FUNCTION_BLOCK FB_SIS_MsgManager_6_0 IMPLEMENTS ITF_MFCS
(**************************************************************************************
 * 	Application		:	BoxControl Framework
 *	Revision		:	$Revision: 404529 $
 *	Revision date	:	$Date: 2018-04-23 08:21:38 +0200 (Mo., 23 Apr 2018) $
 *	Last changed by	:	$Author: b7bolm $
 *	URL				:	$URL: http://almscdc.swisslog.com/repo/SWPD/Development/BoxControlFramework/20_Release/trunk/01_Software/BCF/BCF/JumpStart/20_Product/10_App/11_Com/10_Lib/10_Conv/12_MFCS/11_SIS/FB_SIS_MsgManager_6_0.TcPOU $
 *
 *	Purpose			:	SIS Manager V6.0
 *
 * ------------------------------------------------------------------------------------
 *	Copyright Swisslog [IP AG], Switzerland. All rights reserved.
 * 
 * ------------------------------------------------------------------------------------
 *	
 * 	Revision History: 
 *
 * 	VERSION			DATE			INITIALS			DESCRIPTION
 *	0.1				01.01.2001		swl					Example
 *
 **************************************************************************************)
VAR_INPUT
	Config				: ST_CFG_SIS_MsgManager_6_0; // Configuration
END_VAR

VAR
	Init				: BOOL := FALSE; // Instance initialized	
	RecvTelegram		: ARRAY [1..MAX_APP_DATA_LENGTH] OF BYTE; // Last telegram read from base drive
	SendTelegram		: ARRAY [1..MAX_APP_DATA_LENGTH] OF BYTE; // Last telegram read from base drive
	fbDebugMsg			: FB_DebugMsg; // Debug Messages
	DebugMsg			: STRING(MAX_STRING_LENGTH); // String to compose the logmessage
	fbBaseDriver		: FB_SIS_BaseDriver; // Base SIS driver
	TelegramType		: STRING(3); // SIS Telegram type from the incoming message
	eMsgType			: E_ITC_MsgTypeConv;
	ReceivedLength		: UDINT; // Received length
	WritePointer		: UDINT; // Write pointer to assembly data
	
	TTA					: ST_TTA_6_0; // Struct TTA IN
	TTA_ITC				: ST_ITC_TTA; // Struct TTA IN
	TDQ					: ST_TDQ_6_0; // Struct TDQ IN
	TDQ_ITC				: ST_ITC_TDQ; // Struct TDQ IN
	SCQ					: ST_SCQ_6_0; // Struct SCQ IN
	SCQ_ITC				: ST_ITC_SCQ; // Struct SCQ IN
	GCQ					: ST_GCQ_6_0; // Struct GCQ IN
	GCQ_ITC				: ST_ITC_GCQ; // Struct ECQ IN
	ECQ					: ST_ECQ_6_0; // Struct ECQ IN
	ECQ_ITC				: ST_ITC_ECQ; // Struct ECQ IN
	FCQ					: ST_FCQ_6_0; // Struct FCQ IN
	FCQ_ITC				: ST_ITC_FCQ; // Struct FCQ IN
	SSQ					: ST_SSQ_6_0; // Struct SSQ IN
	SSQ_ITC				: ST_ITC_SSQ; // Struct SSQ IN
	GSQ					: ST_GSQ_6_0; // Struct GSQ IN
	GSQ_ITC				: ST_ITC_GSQ; // Struct GSQ IN
	ESQ					: ST_ESQ_6_0; // Struct ESQ IN
	ESQ_ITC				: ST_ITC_ESQ; // Struct ESQ IN
	FSQ					: ST_FSQ_6_0; // Struct FSQ IN
	FSQ_ITC				: ST_ITC_FSQ; // Struct FSQ IN
	TUQ					: ST_TUQ_6_0; // Struct TUQ IN
	TUQ_ITC				: ST_ITC_TUQ; // Struct TUQ IN
	SIQ					: ST_SIQ_6_0; // Struct SIQ IN
	SIQ_ITC				: ST_ITC_SIQ; // Struct SIQ IN
	MCQ					: ST_MCQ_6_0; // Struct MCQ IN
	MCQ_ITC				: ST_ITC_MCQ; // Struct MCQ IN
	DIQ					: ST_DIQ_6_0; // Struct DIQ IN
	DIQ_ITC				: ST_ITC_DIQ; // Struct DIQ IN
	SDO					: ST_SDO_6_0; // Struct SDO IN
	SDO_ITC				: ST_ITC_SDO; // Struct SDO IN
	IRQ					: ST_IRQ_6_0; // Struct IRQ IN
	IRQ_ITC				: ST_ITC_IRQ; // Struct IRQ IN
	GVQ					: ST_GVQ_6_0; // Struct GVQ IN
	GVQ_ITC				: ST_ITC_GVQ; // Struct GVQ IN
	ECR					: ST_ECR_6_0; // Struct ECR OUT
	ECR_ITC				: ST_ITC_ECR; // Struct ECR OUT
	ESR					: ST_ESR_6_0; // Struct ESR OUT
	ESR_ITC				: ST_ITC_ESR; // Struct ESR ITC
	GCR					: ST_GCR_6_0; // Struct GCR OUT
	GCR_ITC				: ST_ITC_GCR; // Struct GCR ITC
	GSR					: ST_GSR_6_0; // Struct GSR OUT
	GSR_ITC				: ST_ITC_GSR; // Struct GSR ITC
	GVR					: ST_GVR_6_0; // Struct GVR OUT
	GVR_ITC				: ST_ITC_GVR; // Struct GVR ITC
	IPR					: ST_IPR_6_0; // Struct IPR OUT
	IPR_ITC				: ST_ITC_IPR; // Struct IPR ITC
	ISR					: ST_ISR_6_0; // Struct ISR OUT
	ISR_ITC				: ST_ITC_ISR; // Struct ISR ITC
	MCR					: ST_MCR_6_0; // Struct MCR OUT
	MCR_ITC				: ST_ITC_MCR; // Struct MCR ITC
	POR					: ST_POR_6_0; // Struct POR OUT
	POR_ITC				: ST_ITC_POR; // Struct POR ITC
	SCR					: ST_SCR_6_0; // Struct SCR OUT
	SCR_ITC				: ST_ITC_SCR; // Struct SCR ITC
	SDI					: ST_SDI_6_0; // Struct SDI OUT
	SDI_ITC				: ST_ITC_SDI; // Struct SDI ITC
	SIR					: ST_SIR_6_0; // Struct SIR OUT
	SIR_ITC				: ST_ITC_SIR; // Struct SIR ITC
	SNR					: ST_SNR_6_0; // Struct SNR OUT
	SNR_ITC				: ST_ITC_SNR; // Struct SNR ITC
	SSR					: ST_SSR_6_0; // Struct SSR OUT
	SSR_ITC				: ST_ITC_SSR; // Struct SSR ITC
	TDR					: ST_TDR_6_0; // Struct TDR OUT
	TDR_ITC				: ST_ITC_TDR; // Struct TDR ITC
	TTC					: ST_TTC_6_0; // Struct TTC OUT
	TTC_ITC				: ST_ITC_TTC; // Struct TTC ITC
	TTQ					: ST_TTQ_6_0; // Struct TTQ OUT
	TTQ_ITC				: ST_ITC_TTQ; // Struct TTQ ITC
	TUR					: ST_TUR_6_0; // Struct TUR OUT
	TUR_ITC				: ST_ITC_TUR; // Struct TUR ITC
	FSR					: ST_FSR_6_0; // Struct FSR OUT
	FSR_ITC				: ST_ITC_FSR; // Struct FSR ITC
	FCR					: ST_FCR_6_0; // Struct FCR OUT
	FCR_ITC				: ST_ITC_FCR; // Struct FCR ITC
	ATR					: ST_ATR_6_0; // Struct ATR OUT
	ATR_ITC				: ST_ITC_ATR; // Struct ATR ITC
	RTR					: ST_RTR_6_0; // Struct RTR OUT
	RTR_ITC				: ST_ITC_RTR; // Struct RTR ITC
	ERR					: ST_ERR_6_0; // Struct ERR OUT
	ERR_ITC				: ST_ITC_ERR; // Struct ERR ITC
	VIQ					: ST_VIQ_6_0; // Struct VIQ OUT
	VIQ_ITC				: ST_ITC_VIQ; // Struct VIQ ITC
	VIR					: ST_VIR_6_0; // Struct VIR OUT
	VIR_ITC				: ST_ITC_VIR; // Struct VIR ITC
	RAA					: ST_RAA_6_0; // Struct RAA OUT
	RAA_ITC				: ST_ITC_RAA; // Struct RAA ITC
	RAC					: ST_RAC_6_0; // Struct RAC OUT
	RAC_ITC				: ST_ITC_RAC; // Struct RAC OUT
	RDQ					: ST_RDQ_6_0; // Struct RDQ OUT
	RDQ_ITC				: ST_ITC_RDQ; // Struct RDQ OUT
	RDR					: ST_RDR_6_0; // Struct RDR OUT
	RDR_ITC				: ST_ITC_RDR; // Struct RDR ITC
	DAQ					: ST_DAQ_6_0; // Struct DAQ IN
	DAQ_ITC				: ST_ITC_DAQ; // Struct DAQ IN
	GDQ					: ST_GDQ_6_0; // Struct GDQ IN
	GDQ_ITC				: ST_ITC_GDQ; // Struct GDQ IN
	DAR					: ST_DAR_6_0; // Struct DAR OUT
	DAR_ITC				: ST_ITC_DAR; // Struct DAR ITC
	GDR					: ST_GDR_6_0; // Struct GDR OUT
	GDR_ITC				: ST_ITC_GDR; // Struct GDR ITC
	
	
	ECR_String			: T_MaxString; // String
	ESR_String			: T_MaxString; // String
	GCR_String			: T_MaxString; // String
	GSR_String			: T_MaxString; // String
	GVR_String			: T_MaxString; // String
	IPR_String			: T_MaxString; // String
	ISR_String			: T_MaxString; // String
	MCR_String			: T_MaxString; // String
	POR_String			: T_MaxString; // String
	SCR_String			: T_MaxString; // String
	SDI_String			: T_MaxString; // String
	SIR_String			: T_MaxString; // String
	SNR_String			: T_MaxString; // String
	SSR_String			: T_MaxString; // String
	TDR_String			: T_MaxString; // String
	TTC_String			: T_MaxString; // String
	TTQ_String			: T_MaxString; // String
	TUR_String			: T_MaxString; // String
	FSR_String			: T_MaxString; // String
	FCR_String			: T_MaxString; // String
	ATR_String			: T_MaxString; // String
	RTR_String			: T_MaxString; // String
	ERR_String			: T_MaxString; // String
	VIR_String			: T_MaxString; // String
	DAR_String			: T_MaxString; // String
	GDR_String			: T_MaxString; // String
	
	// Robot telegrams
	RCQ_String			: T_MaxString; // String
	RCA_String			: T_MaxString; // String
	RCC_String			: T_MaxString; // String
	RDQ_String			: T_MaxString; // String
	RDR_String			: T_MaxString; // String
	
	Idx					: INT; // Iterator
	TempInt				: INT; // Temporary integer
	IdxOffset			: INT; // Offset telegram length
	NoError				: BOOL; // Temporary no error bit
	BufferWarningActive : BOOL; // Buffer warning level active
	BufferAlarmActive 	: BOOL; // Buffer alarm level active
END_VAR

VAR PERSISTENT
	Settings			: ST_CFG_SIS_MsgManager_6_0; // Active configuration
END_VAR

VAR CONSTANT
	MAX_APP_DATA_LENGTH	: UDINT := 30000;
END_VAR

(**************************************************************************************************************
   SIS Manager - Body never called!
***************************************************************************************************************)
;

ACTION A_PutDAQ:
(**************************************************************************************
 * 	NAME		A_PutDAQ
 * 	FUNCTION	Process DAQ
 **************************************************************************************)

// Clear data structure 
MEMSET(destAddr := ADR(DAQ), fillByte := 0, n := SIZEOF(DAQ));
				
// Copy the TDQ data fields to the DAQ data structure 
IdxOffset := SIS_6_0.APP_DATA_OFFSET+1;
// Copy
MEMCPY(destAddr := ADR(DAQ.Position), srcAddr := ADR(RecvTelegram[IdxOffset]), n := INT_TO_UDINT(SIS_6_0.POSITION_STRINGLENGTH));
// Adjust index
IdxOffset := IdxOffset + SIS_6_0.POSITION_STRINGLENGTH;
// Copy
MEMCPY(destAddr := ADR(DAQ.NumberOfSets), srcAddr := ADR(RecvTelegram[IdxOffset]), n := INT_TO_UDINT(SIS_6_0.DATA_ACQUISITION_NUMBEROFSETS));
// Adjust index
IdxOffset := IdxOffset + SIS_6_0.DATA_ACQUISITION_NUMBEROFSETS;
// Copy
MEMCPY(destAddr := ADR(DAQ.Code), srcAddr := ADR(RecvTelegram[IdxOffset]), n := INT_TO_UDINT(SIS_6_0.DATA_ACQUISITION_CODE));
// Adjust index
IdxOffset := IdxOffset + SIS_6_0.DATA_ACQUISITION_CODE;

FOR Idx := 1 TO STRING_TO_INT(DAQ.NumberOfSets) DO
	
	MEMCPY(destAddr := ADR(DAQ.Variable[Idx]), srcAddr := ADR(RecvTelegram[IdxOffset]), n := INT_TO_UDINT(SIS_6_0.DATA_ACQUISITION_VARIABLENAME));
 
	IdxOffset := IdxOffset + SIS_6_0.DATA_ACQUISITION_VARIABLENAME;
	// Copy
	MEMCPY(destAddr := ADR(DAQ.MaxReportTime[Idx]), srcAddr := ADR(RecvTelegram[IdxOffset]), n := INT_TO_UDINT(SIS_6_0.DATA_ACQUISITION_MAXREPORTTIME));
   // Adjust index
	IdxOffset := IdxOffset + SIS_6_0.DATA_ACQUISITION_MAXREPORTTIME;
	// Copy
	MEMCPY(destAddr := ADR(DAQ.SampleTime[Idx]), srcAddr := ADR(RecvTelegram[IdxOffset]), n := INT_TO_UDINT(SIS_6_0.DATA_ACQUISITION_SAMPLETIME));
	 // Adjust index
	IdxOffset := IdxOffset + SIS_6_0.DATA_ACQUISITION_SAMPLETIME;
	// Copy
	MEMCPY(destAddr := ADR(DAQ.Threshold[Idx]), srcAddr := ADR(RecvTelegram[IdxOffset]), n := INT_TO_UDINT(SIS_6_0.DATA_ACQUISITION_THRESHOLD));
	 // Adjust index
	IdxOffset := IdxOffset + SIS_6_0.DATA_ACQUISITION_THRESHOLD;
	// Copy
	MEMCPY(destAddr := ADR(DAQ.Option[Idx]), srcAddr := ADR(RecvTelegram[IdxOffset]), n := INT_TO_UDINT(SIS_6_0.DATA_ACQUISITION_BIT));
	 // Adjust index
	IdxOffset := IdxOffset + SIS_6_0.DATA_ACQUISITION_BIT;
	// Copy
	MEMCPY(destAddr := ADR(DAQ.Enable[Idx]), srcAddr := ADR(RecvTelegram[IdxOffset]), n := INT_TO_UDINT(SIS_6_0.DATA_ACQUISITION_BIT));
	
	IdxOffset := IdxOffset + SIS_6_0.DATA_ACQUISITION_BIT;
	
END_FOR



// Map to ITC
DAQ_ITC.Position :=  DAQ.Position;
DAQ_ITC.Code := STRING_TO_INT(DAQ.Code);
DAQ_ITC.NumberOfSets := STRING_TO_INT(DAQ.NumberOfSets);

FOR Idx := 1 TO STRING_TO_INT(DAQ.NumberOfSets) DO

	DAQ_ITC.Set[Idx].mVariableName := DAQ.Variable[Idx];
	DAQ_ITC.Set[Idx].MaxReportTime := F_MaxReportTime_TO_Time(sTimeIn:= DAQ.MaxReportTime[Idx]);
	DAQ_ITC.Set[Idx].SampleTime := F_SampleTime_TO_TIME(SampleTimeString:=DAQ.SampleTime[Idx]);
	DAQ_ITC.Set[Idx].Threshold := STRING_TO_INT(DAQ.Threshold[Idx]);
	DAQ_ITC.Set[Idx].Option := INT_TO_BOOL(STRING_TO_INT(DAQ.Option[Idx]));
	DAQ_ITC.Set[Idx].Enable :=  INT_TO_BOOL(STRING_TO_INT(DAQ.Enable[Idx]));
END_FOR

// Forward to mirror channel
M_MirrorData(Data := ADR(RecvTelegram), DataLen := ReceivedLength);

// Forward message to ITC
NoError := fbITC_Manager.M_AddData(
			meChannelSrc := Settings.MFCS_Channel,
			mMsgType	 := E_ITC_MsgTypeConv.DATA_ACQUISITION_REQUEST,
			mpData		 := ADR(DAQ_ITC),
			mLen		 := SIZEOF(DAQ_ITC));

// If forwarding was successful
IF NoError THEN
	// Message processed
	fbBaseDriver.M_ProcessedMsg();
ELSE	
	DebugMsg := 'DAQ - Could not be forwarded to ITC';
	fbDebugMsg.M_SendErrorMsg(DebugMsg);		
END_IF
END_ACTION

ACTION A_PutDIQ:
(**************************************************************************************
 * 	NAME		A_PutDIQ
 * 	FUNCTION	Process DIQ
 **************************************************************************************)
 
// Clear structure
MEMSET(destAddr := ADR(DIQ), fillByte := 0, n := SIZEOF(DIQ));

// Forward to mirror channel
M_MirrorData(Data := ADR(RecvTelegram), DataLen := ReceivedLength);

// Forward message to ITC
NoError := fbITC_Manager.M_AddData(
			meChannelSrc := Settings.MFCS_Channel,
			mMsgType	 := E_ITC_MsgTypeConv.DIGITAL_INPUT_REQUEST,
			mpData		 := 0,
			mLen		 := 0);

// If forwarding was successful
IF NoError THEN
	// Message processed
	fbBaseDriver.M_ProcessedMsg();
	
ELSE	
	DebugMsg := 'DIQ - Could not be forwarded to ITC';
	fbDebugMsg.M_SendErrorMsg(DebugMsg);	
END_IF
END_ACTION

ACTION A_PutECQ:
(**************************************************************************************
 * 	NAME		A_PutECQ
 * 	FUNCTION	Process ECQ
 **************************************************************************************)
 
// Clear data structure 
MEMSET(destAddr := ADR(ECQ), fillByte := 0, n := SIZEOF(ECQ));

// Copy the ECQ data fields to the ECQ data structure 
IdxOffset := SIS_6_0.APP_DATA_OFFSET + 1;

// Copy
MEMCPY(destAddr := ADR(ECQ.Position), srcAddr := ADR(RecvTelegram[IdxOffset]), n := INT_TO_UDINT(SIS_6_0.POSITION_STRINGLENGTH));
// Adjust index
IdxOffset := IdxOffset + SIS_6_0.POSITION_STRINGLENGTH;
// Copy
MEMCPY(destAddr := ADR(ECQ.Code), srcAddr := ADR(RecvTelegram[IdxOffset]), n := INT_TO_UDINT(SIS_6_0.CONTROLCODE_STRINGLENGTH));
// Adjust index
IdxOffset := IdxOffset + SIS_6_0.CONTROLCODE_STRINGLENGTH;
// Copy
MEMCPY(destAddr := ADR(ECQ.Variable), srcAddr := ADR(RecvTelegram[IdxOffset]), n := INT_TO_UDINT(SIS_6_0.CONTROLVARIABLE_STRINGLENGTH));


// Map to ITC
ECQ_ITC.Position := ECQ.Position;
ECQ_ITC.Code := STRING_TO_INT(ECQ.Code);
ECQ_ITC.Variable := STRING_TO_INT(ECQ.Variable);

// Forward to mirror channel
M_MirrorData(Data := ADR(RecvTelegram), DataLen := ReceivedLength);

// Forward message to ITC
NoError := fbITC_Manager.M_AddData(
			meChannelSrc := Settings.MFCS_Channel,
			mMsgType	 := E_ITC_MsgTypeCOnv.ELEMENT_CONTROL_REQUEST,
			mpData		 := ADR(ECQ_ITC),
			mLen		 := SIZEOF(ECQ_ITC));

	
// If forwarding was successful
IF NoError THEN
	// Message processed
	fbBaseDriver.M_ProcessedMsg();
ELSE	
	DebugMsg := 'ECQ - Could not be forwarded to ITC';
	fbDebugMsg.M_SendErrorMsg(DebugMsg);	
END_IF
END_ACTION

ACTION A_PutESQ:
(**************************************************************************************
 * 	NAME		A_PutESQ
 * 	FUNCTION	Process ESQ
 **************************************************************************************)

// Clear data structure 
MEMSET(destAddr := ADR(ESQ), fillByte := 0, n := SIZEOF(ESQ));

// Copy the ESQ data fields to the ESQ data structure 
IdxOffset := SIS_6_0.APP_DATA_OFFSET + 1;

MEMCPY(destAddr := ADR(ESQ.Position), srcAddr := ADR(RecvTelegram[IdxOffset]), n := 12);

// Map to ITC
ESQ_ITC.Position := ESQ.Position;

// Forward to mirror channel
M_MirrorData(Data := ADR(RecvTelegram), DataLen := ReceivedLength);

// Forward message to ITC
NoError := fbITC_Manager.M_AddData(
			meChannelSrc := Settings.MFCS_Channel,
			mMsgType	 := E_ITC_MsgTypeCOnv.ELEMENT_STATUS_REQUEST,
			mpData		 := ADR(ESQ_ITC),
			mLen		 := SIZEOF(ESQ_ITC));

// If forwarding was successful
IF NoError THEN
	// Message processed
	fbBaseDriver.M_ProcessedMsg();
	
ELSE	
	DebugMsg := 'ESQ - Could not be forwarded to ITC';
	fbDebugMsg.M_SendErrorMsg(DebugMsg);
END_IF
END_ACTION

ACTION A_PutFCQ:
(**************************************************************************************
 * 	NAME		A_PutFCQ
 * 	FUNCTION	Process FCQ
 **************************************************************************************)
 
// Clear data structure 
MEMSET(destAddr := ADR(FCQ), fillByte := 0, n := SIZEOF(FCQ));

// Copy the FCQ data fields to the FCQ data structure 
IdxOffset := SIS_6_0.APP_DATA_OFFSET + 1;

// Copy
MEMCPY(destAddr := ADR(FCQ.Position), srcAddr := ADR(RecvTelegram[IdxOffset]), n := INT_TO_UDINT(SIS_6_0.POSITION_STRINGLENGTH));
// Adjust index
IdxOffset := IdxOffset + SIS_6_0.POSITION_STRINGLENGTH;
// Copy
MEMCPY(destAddr := ADR(FCQ.Code), srcAddr := ADR(RecvTelegram[IdxOffset]), n := INT_TO_UDINT(SIS_6_0.CONTROLCODE_STRINGLENGTH));
// Adjust index
IdxOffset := IdxOffset + SIS_6_0.CONTROLCODE_STRINGLENGTH;
// Copy
MEMCPY(destAddr := ADR(FCQ.Variable), srcAddr := ADR(RecvTelegram[IdxOffset]), n := INT_TO_UDINT(SIS_6_0.CONTROLVARIABLE_STRINGLENGTH));

// Map to ITC
FCQ_ITC.Position := FCQ.Position; 
FCQ_ITC.Code := STRING_TO_INT(FCQ.Code);
FCQ_ITC.Variable := STRING_TO_DINT(FCQ.Variable);

// Forward to mirror channel
M_MirrorData(Data := ADR(RecvTelegram), DataLen := ReceivedLength);

// Forward message to ITC
NoError := fbITC_Manager.M_AddData(
			meChannelSrc := Settings.MFCS_Channel,
			mMsgType	 := E_ITC_MsgTypeCOnv.FUNCTION_CONTROL_REQUEST,
			mpData		 := ADR(FCQ_ITC),
			mLen		 := SIZEOF(FCQ_ITC));
	
// If forwarding was successful
IF NoError THEN
	// Message processed
	fbBaseDriver.M_ProcessedMsg();
	
ELSE	
	DebugMsg := 'FCQ - Could not be forwarded to ITC';
	fbDebugMsg.M_SendErrorMsg(DebugMsg);
END_IF
END_ACTION

ACTION A_PutFSQ:
(**************************************************************************************
 * 	NAME		A_PutFSQ
 * 	FUNCTION	Process FSQ
 **************************************************************************************)

// Clear data structure 
MEMSET(destAddr := ADR(FSQ), fillByte := 0, n := SIZEOF(FSQ));

// Copy the FSQ data fields to the FSQ data structure 
IdxOffset := SIS_6_0.APP_DATA_OFFSET + 1;
// Copy
MEMCPY(destAddr := ADR(FSQ.Position), srcAddr := ADR(RecvTelegram[IdxOffset]), n := INT_TO_UDINT(SIS_6_0.POSITION_STRINGLENGTH));

// Map to ITC
FSQ_ITC.Position := FSQ.Position; 

// Forward to mirror channel
M_MirrorData(Data := ADR(RecvTelegram), DataLen := ReceivedLength);

// Forward message to ITC
NoError := fbITC_Manager.M_AddData(
			meChannelSrc := Settings.MFCS_Channel,
			mMsgType	 := E_ITC_MsgTypeCOnv.FUNCTION_STATUS_REQUEST,
			mpData		 := ADR(FSQ_ITC),
			mLen		 := SIZEOF(FSQ_ITC));

// If forwarding was successful
IF NoError THEN
	// Message processed
	fbBaseDriver.M_ProcessedMsg();
	
ELSE	
	DebugMsg := 'FSQ - Could not be forwarded to ITC';
	fbDebugMsg.M_SendErrorMsg(DebugMsg);	
END_IF
END_ACTION

ACTION A_PutGCQ:
(**************************************************************************************
 * 	NAME		A_PutGCQ
 * 	FUNCTION	Process GCQ
 **************************************************************************************)
 
// Clear data structure 
MEMSET(destAddr := ADR(GCQ), fillByte := 0, n := SIZEOF(GCQ));

// Copy the GCQ data fields to the GCQ data structure 
IdxOffset := SIS_6_0.APP_DATA_OFFSET + 1;
// Copy
MEMCPY(destAddr := ADR(GCQ.GroupName), srcAddr := ADR(RecvTelegram[IdxOffset]), n := INT_TO_UDINT(SIS_6_0.POSITION_STRINGLENGTH));
// Adjust index
IdxOffset := IdxOffset + SIS_6_0.POSITION_STRINGLENGTH;
// Copy
MEMCPY(destAddr := ADR(GCQ.Code), srcAddr := ADR(RecvTelegram[IdxOffset]), n := INT_TO_UDINT(SIS_6_0.CONTROLCODE_STRINGLENGTH));
// Adjust index
IdxOffset := IdxOffset + SIS_6_0.CONTROLCODE_STRINGLENGTH;
// Copy
MEMCPY(destAddr := ADR(GCQ.Variable), srcAddr := ADR(RecvTelegram[IdxOffset]), n := INT_TO_UDINT(SIS_6_0.CONTROLVARIABLE_STRINGLENGTH));

// Map to ITC
GCQ_ITC.Position := GCQ.GroupName;
GCQ_ITC.Code := STRING_TO_INT(GCQ.Code);
GCQ_ITC.Variable := STRING_TO_DINT(GCQ.Variable);

// Forward to mirror channel
M_MirrorData(Data := ADR(RecvTelegram), DataLen := ReceivedLength);

// Forward message to ITC
NoError := fbITC_Manager.M_AddData(
			meChannelSrc := Settings.MFCS_Channel,
			mMsgType	 := E_ITC_MsgTypeConv.GROUP_CONTROL_REQUEST,
			mpData		 := ADR(GCQ_ITC),
			mLen		 := SIZEOF(GCQ_ITC));

// If forwarding was successful
IF NoError THEN
	// Message processed
	fbBaseDriver.M_ProcessedMsg();
	
ELSE	
	DebugMsg := 'GCQ - Could not be forwarded to ITC';
	fbDebugMsg.M_SendErrorMsg(DebugMsg);	
END_IF
END_ACTION

ACTION A_PutGDQ:
(**************************************************************************************
 * 	NAME		A_PutGDQ
 * 	FUNCTION	Process GDQ
 **************************************************************************************)

// Clear data structure 
MEMSET(destAddr := ADR(GDQ), fillByte := 0, n := SIZEOF(GDQ));

// Copy the GDQ data fields to the GDQ data structure 
IdxOffset := SIS_6_0.APP_DATA_OFFSET+1;
// Copy
MEMCPY(destAddr := ADR(GDQ.Position), srcAddr := ADR(RecvTelegram[IdxOffset]), n := INT_TO_UDINT(SIS_6_0.POSITION_STRINGLENGTH));
// Adjust index
IdxOffset := IdxOffset + SIS_6_0.POSITION_STRINGLENGTH;
// Copy
MEMCPY(destAddr := ADR(GDQ.Variable), srcAddr := ADR(RecvTelegram[IdxOffset]), n := INT_TO_UDINT(SIS_6_0.DATA_ACQUISITION_VARIABLENAME));
// Adjust index
IdxOffset := IdxOffset + SIS_6_0.DATA_ACQUISITION_VARIABLENAME;

// Map to ITC
GDQ_ITC.Position :=  GDQ.Position;
GDQ_ITC.Variable :=  GDQ.Variable;

// Forward to mirror channel
M_MirrorData(Data := ADR(RecvTelegram), DataLen := ReceivedLength);

// Forward message to ITC
NoError := fbITC_Manager.M_AddData(
			meChannelSrc := Settings.MFCS_Channel,
			mMsgType	 := E_ITC_MsgTypeConv.GATHERED_DATA_REQUEST,
			mpData		 := ADR(GDQ_ITC),
			mLen		 := SIZEOF(GDQ_ITC));

// If forwarding was successful
IF NoError THEN
	// Message processed
	fbBaseDriver.M_ProcessedMsg();
	
ELSE	
	DebugMsg := 'GDQ - Could not be forwarded to ITC';
	fbDebugMsg.M_SendErrorMsg(DebugMsg);	
END_IF
END_ACTION

ACTION A_PutGSQ:
(**************************************************************************************
 * 	NAME		A_PutGSQ
 * 	FUNCTION	Process GSQ
 **************************************************************************************)

// Clear data structure 
MEMSET(destAddr := ADR(GSQ), fillByte := 0, n := SIZEOF(GSQ));

// Copy the GSQ data fields to the GSQ data structure 
IdxOffset := SIS_6_0.APP_DATA_OFFSET + 1;

MEMCPY(destAddr := ADR(GSQ.GroupName), srcAddr := ADR(RecvTelegram[IdxOffset]), n := INT_TO_UDINT(SIS_6_0.POSITION_STRINGLENGTH));

// Map to ITC
GSQ_ITC.Position := GSQ.GroupName;

// Forward to mirror channel
M_MirrorData(Data := ADR(RecvTelegram), DataLen := ReceivedLength);

// Forward message to ITC
NoError := fbITC_Manager.M_AddData(
			meChannelSrc := Settings.MFCS_Channel,
			mMsgType	 := E_ITC_MsgTypeConv.GROUP_STATUS_REQUEST,
			mpData		 := ADR(GSQ_ITC),
			mLen		 := SIZEOF(GSQ_ITC));

// If forwarding was successful
IF NoError THEN
	// Message processed
	fbBaseDriver.M_ProcessedMsg();
	
ELSE	
	DebugMsg := 'GSQ - Could not be forwarded to ITC';
	fbDebugMsg.M_SendErrorMsg(DebugMsg);	
END_IF
END_ACTION

ACTION A_PutGVQ:
(**************************************************************************************
 * 	NAME		A_PutGVQ
 * 	FUNCTION	Process GVQ
 **************************************************************************************)

// Clear data structure 
MEMSET(destAddr := ADR(GVQ), fillByte := 0, n := SIZEOF(GVQ));

// Copy the GVQ data fields to the GVQ data structure 
IdxOffset := SIS_6_0.APP_DATA_OFFSET + 1;
// Copy
MEMCPY(destAddr := ADR(GVQ.Code), srcAddr := ADR(RecvTelegram[IdxOffset]), n := INT_TO_UDINT(SIS_6_0.GVQ_CODE_STRINGLENGTH));
// Adjust index
IdxOffset := IdxOffset + SIS_6_0.GVQ_CODE_STRINGLENGTH;
// Copy
MEMCPY(destAddr := ADR(GVQ.Number), srcAddr := ADR(RecvTelegram[IdxOffset]), n := INT_TO_UDINT(SIS_6_0.GVQ_NUMBER_STRINGLENGTH));
// Adjust index
IdxOffset := IdxOffset + SIS_6_0.GVQ_NUMBER_STRINGLENGTH;
// Copy
MEMCPY(destAddr := ADR(GVQ.Quantity), srcAddr := ADR(RecvTelegram[IdxOffset]), n := INT_TO_UDINT(SIS_6_0.GVQ_QUANTITY_STRINGLENGTH));
// Adjust index
IdxOffset := IdxOffset + SIS_6_0.GVQ_QUANTITY_STRINGLENGTH;
// Copy
MEMCPY(destAddr := ADR(GVQ.Variable[0]), srcAddr := ADR(RecvTelegram[IdxOffset]), n := INT_TO_UDINT(SIS_6_0.GVQ_VARIABLE_STRINGLENGTH));
// Adjust index
IdxOffset := IdxOffset + SIS_6_0.GVQ_VARIABLE_STRINGLENGTH;
// Copy
MEMCPY(destAddr := ADR(GVQ.Variable[1]), srcAddr := ADR(RecvTelegram[IdxOffset]), n := INT_TO_UDINT(SIS_6_0.GVQ_VARIABLE_STRINGLENGTH));
// Adjust index
IdxOffset := IdxOffset + SIS_6_0.GVQ_VARIABLE_STRINGLENGTH;
// Copy
MEMCPY(destAddr := ADR(GVQ.Variable[2]), srcAddr := ADR(RecvTelegram[IdxOffset]), n := INT_TO_UDINT(SIS_6_0.GVQ_VARIABLE_STRINGLENGTH));
// Adjust index
IdxOffset := IdxOffset + SIS_6_0.GVQ_VARIABLE_STRINGLENGTH;
// Copy
MEMCPY(destAddr := ADR(GVQ.Variable[3]), srcAddr := ADR(RecvTelegram[IdxOffset]), n := INT_TO_UDINT(SIS_6_0.GVQ_VARIABLE_STRINGLENGTH));
// Adjust index
IdxOffset := IdxOffset + SIS_6_0.GVQ_VARIABLE_STRINGLENGTH;
// Copy
MEMCPY(destAddr := ADR(GVQ.Variable[4]), srcAddr := ADR(RecvTelegram[IdxOffset]), n := INT_TO_UDINT(SIS_6_0.GVQ_VARIABLE_STRINGLENGTH));
// Adjust index
IdxOffset := IdxOffset + SIS_6_0.GVQ_VARIABLE_STRINGLENGTH;
// Copy
MEMCPY(destAddr := ADR(GVQ.Variable[5]), srcAddr := ADR(RecvTelegram[IdxOffset]), n := INT_TO_UDINT(SIS_6_0.GVQ_VARIABLE_STRINGLENGTH));
// Adjust index
IdxOffset := IdxOffset + SIS_6_0.GVQ_VARIABLE_STRINGLENGTH;
// Copy
MEMCPY(destAddr := ADR(GVQ.Variable[6]), srcAddr := ADR(RecvTelegram[IdxOffset]), n := INT_TO_UDINT(SIS_6_0.GVQ_VARIABLE_STRINGLENGTH));
// Adjust index
IdxOffset := IdxOffset + SIS_6_0.GVQ_VARIABLE_STRINGLENGTH;
// Copy
MEMCPY(destAddr := ADR(GVQ.Variable[7]), srcAddr := ADR(RecvTelegram[IdxOffset]), n := INT_TO_UDINT(SIS_6_0.GVQ_VARIABLE_STRINGLENGTH));
// Adjust index
IdxOffset := IdxOffset + SIS_6_0.GVQ_VARIABLE_STRINGLENGTH;
// Copy
MEMCPY(destAddr := ADR(GVQ.Variable[8]), srcAddr := ADR(RecvTelegram[IdxOffset]), n := INT_TO_UDINT(SIS_6_0.GVQ_VARIABLE_STRINGLENGTH));
// Adjust index
IdxOffset := IdxOffset + SIS_6_0.GVQ_VARIABLE_STRINGLENGTH;
// Copy
MEMCPY(destAddr := ADR(GVQ.Variable[9]), srcAddr := ADR(RecvTelegram[IdxOffset]), n := INT_TO_UDINT(SIS_6_0.GVQ_VARIABLE_STRINGLENGTH));

// Map to ITC
GVQ_ITC.Code := STRING_TO_INT(GVQ.Code);
GVQ_ITC.Number := STRING_TO_INT(GVQ.Number);
GVQ_ITC.Quantity := STRING_TO_INT(GVQ.Quantity);
GVQ_ITC.Variable[0] := STRING_TO_DINT(GVQ.Variable[0]);
GVQ_ITC.Variable[1] := STRING_TO_DINT(GVQ.Variable[1]);
GVQ_ITC.Variable[2] := STRING_TO_DINT(GVQ.Variable[2]);
GVQ_ITC.Variable[3] := STRING_TO_DINT(GVQ.Variable[3]);
GVQ_ITC.Variable[4] := STRING_TO_DINT(GVQ.Variable[4]);
GVQ_ITC.Variable[5] := STRING_TO_DINT(GVQ.Variable[5]);
GVQ_ITC.Variable[6] := STRING_TO_DINT(GVQ.Variable[6]);
GVQ_ITC.Variable[7] := STRING_TO_DINT(GVQ.Variable[7]);
GVQ_ITC.Variable[8] := STRING_TO_DINT(GVQ.Variable[8]);
GVQ_ITC.Variable[9] := STRING_TO_DINT(GVQ.Variable[9]);

// Forward to mirror channel
M_MirrorData(Data := ADR(RecvTelegram), DataLen := ReceivedLength);

// Forward message to ITC
NoError := fbITC_Manager.M_AddData(
			meChannelSrc := Settings.MFCS_Channel,
			mMsgType	 := E_ITC_MsgTypeConv.GLOBAL_VARIABLE_REQUEST,
			mpData		 := ADR(GVQ_ITC),
			mLen	 := SIZEOF(GVQ_ITC));
	
// If forwarding was successful
IF NoError THEN
	// Message processed
	fbBaseDriver.M_ProcessedMsg();
	
ELSE	
	DebugMsg := 'GVQ - Could not be forwarded to ITC';
	fbDebugMsg.M_SendErrorMsg(DebugMsg);	
END_IF
END_ACTION

ACTION A_PutIRQ:
(**************************************************************************************
 * 	NAME		A_PutIRQ
 * 	FUNCTION	Process IRQ
 **************************************************************************************)
 
// Clear data structure 
MEMSET(destAddr := ADR(IRQ), fillByte := 0, n := SIZEOF(IRQ));

// Copy the IRQ data fields to the IRQ data structure 
IdxOffset := SIS_6_0.APP_DATA_OFFSET + 1;
// Copy
MEMCPY(destAddr := ADR(IRQ.SignalType), srcAddr := ADR(RecvTelegram[IdxOffset]), n := INT_TO_UDINT(SIS_6_0.IRQ_SIGNALTYPE_STRINGLENGTH));
// Adjust index
IdxOffset := IdxOffset + SIS_6_0.IRQ_SIGNALTYPE_STRINGLENGTH;
// Copy
MEMCPY(destAddr := ADR(IRQ.StartSignalNumber), srcAddr := ADR(RecvTelegram[IdxOffset]), n := INT_TO_UDINT(SIS_6_0.IRQ_START_SIGNAL_NUMBER_STRINGLENGTH));
// Adjust index
IdxOffset := IdxOffset + SIS_6_0.IRQ_START_SIGNAL_NUMBER_STRINGLENGTH;
// Copy
MEMCPY(destAddr := ADR(IRQ.DataLength), srcAddr := ADR(RecvTelegram[IdxOffset]), n := INT_TO_UDINT(SIS_6_0.IRQ_DATALENGTH_STRINGLENGTH));

// Map to ITC
IRQ_ITC.DataLength := STRING_TO_INT(IRQ.DataLength);
IRQ_ITC.SignalType := STRING_TO_INT(IRQ.SignalType);
IRQ_ITC.StartSignalNumber := STRING_TO_INT(IRQ.StartSignalNumber);

// Forward to mirror channel
M_MirrorData(Data := ADR(RecvTelegram), DataLen := ReceivedLength);

// Forward message to ITC
NoError := fbITC_Manager.M_AddData(
			meChannelSrc := Settings.MFCS_Channel,
			mMsgType	 := E_ITC_MsgTypeConv.I_O_STATUS_REQUEST,
			mpData		 := ADR(IRQ_ITC),
			mLen		 := SIZEOF(IRQ_ITC));


// If forwarding was successful
IF NoError THEN
	// Message processed
	fbBaseDriver.M_ProcessedMsg();
	
ELSE	
	DebugMsg := 'IRQ - Could not be forwarded to ITC';
	fbDebugMsg.M_SendErrorMsg(DebugMsg);	
END_IF
END_ACTION

ACTION A_PutMCQ:
(**************************************************************************************
 * 	NAME		A_PutMCQ
 * 	FUNCTION	Process MCQ
 **************************************************************************************)
 
// Clear data structure 
MEMSET(destAddr := ADR(MCQ), fillByte := 0, n := SIZEOF(MCQ));

// Copy the MCQ data fields to the MCQ data structure 
IdxOffset := SIS_6_0.APP_DATA_OFFSET + 1;
// Copy
MEMCPY(destAddr := ADR(MCQ.Position), srcAddr := ADR(RecvTelegram[IdxOffset]), n := INT_TO_UDINT(SIS_6_0.POSITION_STRINGLENGTH));
// Adjust index
IdxOffset := IdxOffset + SIS_6_0.POSITION_STRINGLENGTH;
// Copy
MEMCPY(destAddr := ADR(MCQ.Code), srcAddr := ADR(RecvTelegram[IdxOffset]), n := INT_TO_UDINT(SIS_6_0.MCQ_CODE_STRINGLENGTH));
// Adjust index
IdxOffset := IdxOffset + SIS_6_0.MCQ_CODE_STRINGLENGTH;
// Copy
MEMCPY(destAddr := ADR(MCQ.Speed), srcAddr := ADR(RecvTelegram[IdxOffset]), n := INT_TO_UDINT(SIS_6_0.MCQ_SPEED_STRINGLENGTH));
// Adjust index
IdxOffset := IdxOffset + SIS_6_0.MCQ_SPEED_STRINGLENGTH;
// Copy
MEMCPY(destAddr := ADR(MCQ.Axis1Fwd), srcAddr := ADR(RecvTelegram[IdxOffset]), n := INT_TO_UDINT(SIS_6_0.MCQ_AXIS_STRINGLENGTH));
// Adjust index
IdxOffset := IdxOffset + SIS_6_0.MCQ_AXIS_STRINGLENGTH;
// Copy
MEMCPY(destAddr := ADR(MCQ.Axis1Rev), srcAddr := ADR(RecvTelegram[IdxOffset]), n := INT_TO_UDINT(SIS_6_0.MCQ_AXIS_STRINGLENGTH));
// Adjust index
IdxOffset := IdxOffset + SIS_6_0.MCQ_AXIS_STRINGLENGTH;
// Copy
MEMCPY(destAddr := ADR(MCQ.Axis2Fwd), srcAddr := ADR(RecvTelegram[IdxOffset]), n :=INT_TO_UDINT(SIS_6_0.MCQ_AXIS_STRINGLENGTH));
// Adjust index
IdxOffset := IdxOffset + SIS_6_0.MCQ_AXIS_STRINGLENGTH;
// Copy
MEMCPY(destAddr := ADR(MCQ.Axis2Rev), srcAddr := ADR(RecvTelegram[IdxOffset]), n := INT_TO_UDINT(SIS_6_0.MCQ_AXIS_STRINGLENGTH));
// Adjust index
IdxOffset := IdxOffset + SIS_6_0.MCQ_AXIS_STRINGLENGTH;
// Copy
MEMCPY(destAddr := ADR(MCQ.Axis3Fwd), srcAddr := ADR(RecvTelegram[IdxOffset]), n := INT_TO_UDINT(SIS_6_0.MCQ_AXIS_STRINGLENGTH));
// Adjust index
IdxOffset := IdxOffset + SIS_6_0.MCQ_AXIS_STRINGLENGTH;
// Copy
MEMCPY(destAddr := ADR(MCQ.Axis3Rev), srcAddr := ADR(RecvTelegram[IdxOffset]), n := INT_TO_UDINT(SIS_6_0.MCQ_AXIS_STRINGLENGTH));
// Adjust index
IdxOffset := IdxOffset + SIS_6_0.MCQ_AXIS_STRINGLENGTH;
// Copy
MEMCPY(destAddr := ADR(MCQ.Axis4Fwd), srcAddr := ADR(RecvTelegram[IdxOffset]), n := INT_TO_UDINT(SIS_6_0.MCQ_AXIS_STRINGLENGTH));
// Adjust index
IdxOffset := IdxOffset + SIS_6_0.MCQ_AXIS_STRINGLENGTH;
// Copy
MEMCPY(destAddr := ADR(MCQ.Axis4Rev), srcAddr := ADR(RecvTelegram[IdxOffset]), n := INT_TO_UDINT(SIS_6_0.MCQ_AXIS_STRINGLENGTH));
// Adjust index
IdxOffset := IdxOffset + SIS_6_0.MCQ_AXIS_STRINGLENGTH;
// Copy
MEMCPY(destAddr := ADR(MCQ.Axis5Fwd), srcAddr := ADR(RecvTelegram[IdxOffset]), n := INT_TO_UDINT(SIS_6_0.MCQ_AXIS_STRINGLENGTH));
// Adjust index
IdxOffset := IdxOffset + SIS_6_0.MCQ_AXIS_STRINGLENGTH;
// Copy
MEMCPY(destAddr := ADR(MCQ.Axis5Rev), srcAddr := ADR(RecvTelegram[IdxOffset]), n := INT_TO_UDINT(SIS_6_0.MCQ_AXIS_STRINGLENGTH));
// Adjust index
IdxOffset := IdxOffset + SIS_6_0.MCQ_AXIS_STRINGLENGTH;
// Copy
MEMCPY(destAddr := ADR(MCQ.Axis6Fwd), srcAddr := ADR(RecvTelegram[IdxOffset]), n := INT_TO_UDINT(SIS_6_0.MCQ_AXIS_STRINGLENGTH));
// Adjust index
IdxOffset := IdxOffset + SIS_6_0.MCQ_AXIS_STRINGLENGTH;
// Copy
MEMCPY(destAddr := ADR(MCQ.Axis6Rev), srcAddr := ADR(RecvTelegram[IdxOffset]), n := INT_TO_UDINT(SIS_6_0.MCQ_AXIS_STRINGLENGTH));
// Adjust index
IdxOffset := IdxOffset + SIS_6_0.MCQ_AXIS_STRINGLENGTH;
// Copy
MEMCPY(destAddr := ADR(MCQ.Button1), srcAddr := ADR(RecvTelegram[IdxOffset]), n := INT_TO_UDINT(SIS_6_0.MCQ_BUTTON_STRINGLENGTH));
// Adjust index
IdxOffset := IdxOffset + SIS_6_0.MCQ_BUTTON_STRINGLENGTH;
// Copy
MEMCPY(destAddr := ADR(MCQ.Button2), srcAddr := ADR(RecvTelegram[IdxOffset]), n := INT_TO_UDINT(SIS_6_0.MCQ_BUTTON_STRINGLENGTH));

// Map to ITC
MCQ_ITC.Position 	:= MCQ.Position;
MCQ_ITC.Code		:= STRING_TO_INT(MCQ.Code);
MCQ_ITC.Speed		:= MCQ.Speed = '1';
MCQ_ITC.Axis1Fwd	:= MCQ.Axis1Fwd = '1';
MCQ_ITC.Axis1Rev	:= MCQ.Axis1Rev = '1';
MCQ_ITC.Axis2Fwd	:= MCQ.Axis2Fwd = '1';
MCQ_ITC.Axis2Rev	:= MCQ.Axis2Rev = '1';
MCQ_ITC.Axis3Fwd	:= MCQ.Axis3Fwd = '1';
MCQ_ITC.Axis3Rev	:= MCQ.Axis3Rev = '1';
MCQ_ITC.Axis4Fwd	:= MCQ.Axis4Fwd = '1';
MCQ_ITC.Axis4Rev	:= MCQ.Axis4Rev = '1';
MCQ_ITC.Axis5Fwd	:= MCQ.Axis5Fwd = '1';
MCQ_ITC.Axis5Rev	:= MCQ.Axis5Rev = '1';
MCQ_ITC.Axis6Fwd	:= MCQ.Axis6Fwd = '1';
MCQ_ITC.Axis6Rev	:= MCQ.Axis6Rev = '1';
MCQ_ITC.Button1		:= MCQ.Button1 = '1';
MCQ_ITC.Button2		:= MCQ.Button2 = '1';

// Forward to mirror channel
M_MirrorData(Data := ADR(RecvTelegram), DataLen := ReceivedLength);

// Forward message to ITC
NoError := fbITC_Manager.M_AddData(
			meChannelSrc := Settings.MFCS_Channel,
			mMsgType	 := E_ITC_MsgTypeConv.MANUAL_CONTROL_REQUEST,
			mpData		 := ADR(MCQ_ITC),
			mLen		 := SIZEOF(MCQ_ITC));

// If forwarding was successful
IF NoError THEN
	// Message processed
	fbBaseDriver.M_ProcessedMsg();
	
ELSE	
	DebugMsg := 'MCQ - Could not be forwarded to ITC';
	fbDebugMsg.M_SendErrorMsg(DebugMsg);	
END_IF
END_ACTION

ACTION A_PutRAA:
(**************************************************************************************
 * 	NAME		A_PutRAA
 * 	FUNCTION	Process RAA
 **************************************************************************************)

// Clear data structure 
MEMSET(destAddr := ADR(RAA), fillByte := 0, n := SIZEOF(RAA));

// Copy the RAA data fields to the RAA data structure 
IdxOffset := SIS_6_0.APP_DATA_OFFSET + 1;
// Copy
MEMCPY(destAddr := ADR(RAA.Position), srcAddr := ADR(RecvTelegram[IdxOffset]), n := INT_TO_UDINT(SIS_6_0.POSITION_STRINGLENGTH));
// Adjust index
IdxOffset := IdxOffset + SIS_6_0.POSITION_STRINGLENGTH;
// Copy
MEMCPY(destAddr := ADR(RAA.CommandDataIndex), srcAddr := ADR(RecvTelegram[IdxOffset]), n := INT_TO_UDINT(SIS_6_0.RAA_COMMAND_DATA_INDEX_STRINGLENGTH));
// Adjust index
IdxOffset := IdxOffset + SIS_6_0.RAA_COMMAND_DATA_INDEX_STRINGLENGTH;
// Copy
MEMCPY(destAddr := ADR(RAA.CommandPriority), srcAddr := ADR(RecvTelegram[IdxOffset]), n := INT_TO_UDINT(SIS_6_0.RAA_COMMAND_PRIORITY_STRINGLENGTH));
// Adjust index
IdxOffset := IdxOffset + SIS_6_0.RAA_COMMAND_PRIORITY_STRINGLENGTH;
// Copy
MEMCPY(destAddr := ADR(RAA.AssignmentID), srcAddr := ADR(RecvTelegram[IdxOffset]), n := INT_TO_UDINT(SIS_6_0.RAA_ASSIGNMENT_ID_STRINGLENGTH));
// Adjust index
IdxOffset := IdxOffset + SIS_6_0.RAA_ASSIGNMENT_ID_STRINGLENGTH;
// Copy
MEMCPY(destAddr := ADR(RAA.CommandSequenceIndex), srcAddr := ADR(RecvTelegram[IdxOffset]), n := INT_TO_UDINT(SIS_6_0.RAA_SEQUENCE_INDEX_STRINGLENGTH));
// Adjust index
IdxOffset := IdxOffset + SIS_6_0.RAA_SEQUENCE_INDEX_STRINGLENGTH;
// Copy
MEMCPY(destAddr := ADR(RAA.CommandSequenceSize), srcAddr := ADR(RecvTelegram[IdxOffset]), n := INT_TO_UDINT(SIS_6_0.RAA_SEQUENCE_SIZE_STRINGLENGTH));
// Adjust index
IdxOffset := IdxOffset + SIS_6_0.RAA_SEQUENCE_SIZE_STRINGLENGTH;
// Copy
MEMCPY(destAddr := ADR(RAA.CommandArgsCount), srcAddr := ADR(RecvTelegram[IdxOffset]), n := INT_TO_UDINT(SIS_6_0.RAA_COMMAND_ARGS_COUNT_STRINGLENGTH));
// Adjust index
IdxOffset := IdxOffset + SIS_6_0.RAA_COMMAND_ARGS_COUNT_STRINGLENGTH;

IF STRING_TO_INT(RAA.CommandArgsCount) <= SIS_6_0.RAA_NUMBER_OF_COMMAND_ARGS THEN
	FOR Idx := 1 TO STRING_TO_INT(RAA.CommandArgsCount) BY 1 DO
		// Copy
		MEMCPY(destAddr := ADR(RAA.CommandArgs[Idx].Key), srcAddr := ADR(RecvTelegram[IdxOffset]), n := INT_TO_UDINT(SIS_6_0.RAA_COMMAND_ARGS_KEY_STRINGLENGTH));
		// Adjust index
		IdxOffset := IdxOffset + SIS_6_0.RAA_COMMAND_ARGS_KEY_STRINGLENGTH;
		// Copy
		MEMCPY(destAddr := ADR(RAA.CommandArgs[Idx].Value), srcAddr := ADR(RecvTelegram[IdxOffset]), n := INT_TO_UDINT(SIS_6_0.RAA_COMMAND_ARGS_VALUE_STRINGLENGTH));
		// Adjust index
		IdxOffset := IdxOffset + SIS_6_0.RAA_COMMAND_ARGS_VALUE_STRINGLENGTH;
	END_FOR
END_IF

// Copy
MEMCPY(destAddr := ADR(RAA.RobotCommand), srcAddr := ADR(RecvTelegram[IdxOffset]), n := INT_TO_UDINT(SIS_6_0.RAA_ROBOT_COMMAND_STRINGLENGTH));

// Map to ITC
RAA_ITC.Position				:= RAA.Position;
RAA_ITC.CommandDataIndex		:= STRING_TO_INT(RAA.CommandDataIndex);
RAA_ITC.CommandPriority			:= STRING_TO_INT(RAA.CommandPriority);
RAA_ITC.AssignmentID			:= STRING_TO_UDINT(RAA.AssignmentID);
RAA_ITC.GroupID					:= STRING_TO_ULINT(RAA.CommandSequenceIndex);
RAA_ITC.LastGroupInSequence		:= STRING_TO_INT(RAA.CommandSequenceSize);
RAA_ITC.CommandArgsCount		:= STRING_TO_DINT(RAA.CommandArgsCount);

FOR Idx := 1 TO STRING_TO_INT(RAA.CommandArgsCount) BY 1 DO 
	RAA_ITC.CommandArgs[Idx].Key	:= RAA.CommandArgs[Idx].Key;
	RAA_ITC.CommandArgs[Idx].Value	:= RAA.CommandArgs[Idx].Value;
END_FOR

RAA_ITC.RobotCommand				:= RAA.RobotCommand;

// Forward to mirror channel
M_MirrorData(Data := ADR(RecvTelegram), DataLen := ReceivedLength);

// Forward message to ITC
NoError := fbITC_Manager.M_AddData(
			meChannelSrc := Settings.MFCS_Channel,
			mMsgType	 := E_ITC_MsgTypeConv.ROBOT_ACTION_ASSIGNMENT,
			mpData		 := ADR(RAA_ITC),
			mLen		 := SIZEOF(RAA_ITC));
			
IF NoError THEN			
	// Message processed
	fbBaseDriver.M_ProcessedMsg();

ELSE	
	DebugMsg := 'RAA - Could not be forwarded to ITC';
	fbDebugMsg.M_SendErrorMsg(DebugMsg);	
END_IF
END_ACTION

ACTION A_PutRDQ:
(**************************************************************************************
 * 	NAME		A_PutRDQ
 * 	FUNCTION	Process RDQ
 **************************************************************************************)

// Clear data structure 
MEMSET(destAddr := ADR(RDQ), fillByte := 0, n := SIZEOF(RDQ));

// Copy the RDQ data fields to the RDQ data structure 
IdxOffset := SIS_6_0.APP_DATA_OFFSET + 1;
// Copy
MEMCPY(destAddr := ADR(RDQ.Position), srcAddr := ADR(RecvTelegram[IdxOffset]), n := INT_TO_UDINT(SIS_6_0.POSITION_STRINGLENGTH));
// Adjust index
IdxOffset := IdxOffset + SIS_6_0.POSITION_STRINGLENGTH;
// Copy
MEMCPY(destAddr := ADR(RDQ.CommandDataIndex), srcAddr := ADR(RecvTelegram[IdxOffset]), n := INT_TO_UDINT(SIS_6_0.RDQ_COMMAND_DATA_INDEX_STRINGLENGTH));
// Adjust index
IdxOffset := IdxOffset + SIS_6_0.RDQ_COMMAND_DATA_INDEX_STRINGLENGTH;
// Copy
MEMCPY(destAddr := ADR(RDQ.AssignmentID), srcAddr := ADR(RecvTelegram[IdxOffset]), n := INT_TO_UDINT(SIS_6_0.ASSIGNMENT_ID_STRINGLENGTH));
// Adjust index
IdxOffset := IdxOffset + SIS_6_0.ASSIGNMENT_ID_STRINGLENGTH;
// Copy
MEMCPY(destAddr := ADR(RDQ.CommandSequenceIndex), srcAddr := ADR(RecvTelegram[IdxOffset]), n := INT_TO_UDINT(SIS_6_0.RDQ_COMMAND_SEQUENCE_INDEX_STRINGLENGTH));
// Adjust index
IdxOffset := IdxOffset + SIS_6_0.RDQ_COMMAND_SEQUENCE_INDEX_STRINGLENGTH;
// Copy
MEMCPY(destAddr := ADR(RDQ.Code), srcAddr := ADR(RecvTelegram[IdxOffset]), n := INT_TO_UDINT(SIS_6_0.ERR_CODE_STRINGLENGTH));
// Adjust index
IdxOffset := IdxOffset + SIS_6_0.ERR_CODE_STRINGLENGTH;

// Map to ITC
RDQ_ITC.Position	 		:= RDQ.Position;
RDQ_ITC.CommandDataIndex	:= STRING_TO_INT(RDQ.CommandDataIndex);
RDQ_ITC.AssignmentID		:= STRING_TO_UDINT(RDQ.AssignmentID);
RDQ_ITC.GroupID				:= STRING_TO_ULINT(RDQ.CommandSequenceIndex);
RDQ_ITC.Code				:= STRING_TO_INT(RDQ.Code);

// Forward to mirror channel
M_MirrorData(Data := ADR(RecvTelegram), DataLen := ReceivedLength);

// Forward message to ITC
NoError := fbITC_Manager.M_AddData(
			meChannelSrc := Settings.MFCS_Channel,
			mMsgType	 := E_ITC_MsgTypeConv.ROBOT_DELETE_REQUEST,
			mpData		 := ADR(RDQ_ITC),
			mLen		 := SIZEOF(RDQ_ITC));
			
IF NoError THEN			
	// Message processed
	fbBaseDriver.M_ProcessedMsg();
ELSE	
	DebugMsg := 'RDQ - Could not be forwarded to ITC';
	fbDebugMsg.M_SendErrorMsg(DebugMsg);	
END_IF
END_ACTION

ACTION A_PutSCQ:
(**************************************************************************************
 * 	NAME		A_PutSCQ
 * 	FUNCTION	Process SCQ
 **************************************************************************************)
 
// Clear data structure 
MEMSET(destAddr := ADR(SCQ), fillByte := 0, n := SIZEOF(SCQ));

// Copy the SCQ data fields to the SCQ data structure 
IdxOffset := SIS_6_0.APP_DATA_OFFSET + 1;
// Copy
MEMCPY(destAddr := ADR(SCQ.SubsystemName), srcAddr := ADR(RecvTelegram[IdxOffset]), n := INT_TO_UDINT(SIS_6_0.POSITION_STRINGLENGTH));
// Adjust index
IdxOffset := IdxOffset + SIS_6_0.POSITION_STRINGLENGTH;
// Copy
MEMCPY(destAddr := ADR(SCQ.Code), srcAddr := ADR(RecvTelegram[IdxOffset]), n := INT_TO_UDINT(SIS_6_0.CONTROLCODE_STRINGLENGTH));
// Adjust index
IdxOffset := IdxOffset + SIS_6_0.CONTROLCODE_STRINGLENGTH;
// Copy
MEMCPY(destAddr := ADR(SCQ.Variable), srcAddr := ADR(RecvTelegram[IdxOffset]), n := INT_TO_UDINT(SIS_6_0.CONTROLVARIABLE_STRINGLENGTH));
// Adjust index
IdxOffset := IdxOffset + SIS_6_0.CONTROLVARIABLE_STRINGLENGTH;
// Copy
MEMCPY(destAddr := ADR(SCQ.SystemTime), srcAddr := ADR(RecvTelegram[IdxOffset]), n := INT_TO_UDINT(SIS_6_0.TIMESTAMP_STRINGLENGTH));
 
// Map to ITC
SCQ_ITC.SubsystemName := SCQ.SubsystemName;
SCQ_ITC.Code := STRING_TO_INT(SCQ.Code);
SCQ_ITC.Variable := STRING_TO_DINT(SCQ.Variable);
SCQ_ITC.SystemTime := SCQ.SystemTime;

// Forward to mirror channel
M_MirrorData(Data := ADR(RecvTelegram), DataLen := ReceivedLength);

// Forward message to ITC
NoError := fbITC_Manager.M_AddData(
			meChannelSrc := Settings.MFCS_Channel,
			mMsgType	 := E_ITC_MsgTypeConv.SUBSYSTEM_CONTROL_REQUEST,
			mpData		 := ADR(SCQ_ITC),
			mLen		 := SIZEOF(SCQ_ITC));

// If forwarding was successful
IF NoError THEN
	// Message processed
	fbBaseDriver.M_ProcessedMsg();
	
ELSE	
	DebugMsg := 'SCQ - Could not be forwarded to ITC';
	fbDebugMsg.M_SendErrorMsg(DebugMsg);	
END_IF
END_ACTION

ACTION A_PutSDO:
(**************************************************************************************
 * 	NAME		A_PutSDO
 * 	FUNCTION	Process SDO
 **************************************************************************************)
 
// Clear data structure 
MEMSET(destAddr := ADR(SDO), fillByte := 0, n := SIZEOF(SDO));

// Copy the SDO data fields to the SDO data structure 
IdxOffset := SIS_6_0.APP_DATA_OFFSET + 1;

// Copy
MEMCPY(destAddr := ADR(SDO.SignalNumber), srcAddr := ADR(RecvTelegram[IdxOffset]), n := INT_TO_UDINT(SIS_6_0.SDO_SIGNAL_NUMBER_STRINGLENGTH));
// Adjust index
IdxOffset := IdxOffset + SIS_6_0.SDO_SIGNAL_NUMBER_STRINGLENGTH;
// Copy
MEMCPY(destAddr := ADR(SDO.SignalState), srcAddr := ADR(RecvTelegram[IdxOffset]), n := INT_TO_UDINT(SIS_6_0.SDO_SIGNALSTATE_STRINGLENGTH));


// Map to ITC
SDO_ITC.SignalNumber := STRING_TO_INT(SDO.SignalNumber);
SDO_ITC.SignalState := STRING_TO_INT(SDO.SignalState);

// Forward to mirror channel
M_MirrorData(Data := ADR(RecvTelegram), DataLen := ReceivedLength);

// Forward message to ITC
NoError := fbITC_Manager.M_AddData(
			meChannelSrc := Settings.MFCS_Channel,
			mMsgType	 := E_ITC_MsgTypeConv.SET_DIGITAL_OUTPUT,
			mpData		 := ADR(SDO_ITC),
			mLen		 := SIZEOF(SDO_ITC));

// If forwarding was successful
IF NoError THEN
	// Message processed
	fbBaseDriver.M_ProcessedMsg();
	
ELSE	
	DebugMsg := 'SDO - Could not be forwarded to ITC';
	fbDebugMsg.M_SendErrorMsg(DebugMsg);	
END_IF
END_ACTION

ACTION A_PutSIQ:
(**************************************************************************************
 * 	NAME		A_PutSIQ
 * 	FUNCTION	Process SIQ
 **************************************************************************************)
 
// Clear data structure 
MEMSET(destAddr := ADR(SIQ), fillByte := 0, n := SIZEOF(SIQ));

// Copy the SIQ data fields to the SIQ data structure 
IdxOffset := SIS_6_0.APP_DATA_OFFSET + 1;

// Copy
MEMCPY(destAddr := ADR(SIQ.Position), srcAddr := ADR(RecvTelegram[IdxOffset]), n := INT_TO_UDINT(SIS_6_0.POSITION_STRINGLENGTH));
// Adjust index
IdxOffset := IdxOffset + SIS_6_0.POSITION_STRINGLENGTH;
// Copy
MEMCPY(destAddr := ADR(SIQ.CODE), srcAddr := ADR(RecvTelegram[IdxOffset]), n := INT_TO_UDINT(SIS_6_0.SIQ_CODE_STRINGLENGTH));

// Map to ITC
SIQ_ITC.Position := SIQ.Position;
SIQ_ITC.Code := STRING_TO_INT(SIQ.Code);

// Forward to mirror channel
M_MirrorData(Data := ADR(RecvTelegram), DataLen := ReceivedLength);

// Forward message to ITC
NoError := fbITC_Manager.M_AddData(
			meChannelSrc := Settings.MFCS_Channel,
			mMsgType	 := E_ITC_MsgTypeConv.SCANNER_INFORMATION_REQUEST,
			mpData		 := ADR(SIQ_ITC),
			mLen		 := SIZEOF(SIQ_ITC));

// If forwarding was successful
IF NoError THEN
	// Message processed
	fbBaseDriver.M_ProcessedMsg();
	
ELSE	
	DebugMsg := 'SIQ - Could not be forwarded to ITC';
	fbDebugMsg.M_SendErrorMsg(DebugMsg);	
END_IF
END_ACTION

ACTION A_PutSSQ:
(**************************************************************************************
 * 	NAME		A_PutSSQ
 * 	FUNCTION	Process SSQ
 **************************************************************************************)
 
// Clear data structure 
MEMSET(destAddr := ADR(SSQ), fillByte := 0, n := SIZEOF(SSQ));

// Copy the SSQ data fields to the PLQ data structure
IdxOffset := SIS_6_0.APP_DATA_OFFSET + 1;
// Copy
MEMCPY(destAddr := ADR(SSQ.SubsystemName), srcAddr := ADR(RecvTelegram[IdxOffset]), n := INT_TO_UDINT(SIS_6_0.POSITION_STRINGLENGTH));


// Map to ITC
SSQ_ITC.Position := SSQ.SubsystemName;

// Forward to mirror channel
M_MirrorData(Data := ADR(RecvTelegram), DataLen := ReceivedLength);

// Forward message to ITC
NoError := fbITC_Manager.M_AddData(
			meChannelSrc := Settings.MFCS_Channel,
			mMsgType	 := E_ITC_MsgTypeConv.SUBSYSTEM_STATUS_REQUEST,
			mpData		 := ADR(SSQ_ITC),
			mLen		 := SIZEOF(SSQ_ITC));

// If forwarding was successful
IF NoError THEN
	// Message processed
	fbBaseDriver.M_ProcessedMsg();
	
ELSE	
	DebugMsg := 'SSQ - Could not be forwarded to ITC';
	fbDebugMsg.M_SendErrorMsg(DebugMsg);	
END_IF
END_ACTION

ACTION A_PutTDQ:
(**************************************************************************************
 * 	NAME		A_PutTDQ
 * 	FUNCTION	Process TDQ
 **************************************************************************************)
 
// Clear data structure 
MEMSET(destAddr := ADR(TDQ), fillByte := 0, n := SIZEOF(TDQ));
				
// Copy the TDQ data fields to the TDQ data structure 
IdxOffset := SIS_6_0.APP_DATA_OFFSET + 1;
// Copy
MEMCPY(destAddr := ADR(TDQ.Position), srcAddr := ADR(RecvTelegram[IdxOffset]), n := INT_TO_UDINT(SIS_6_0.POSITION_STRINGLENGTH));
// Adjust index
IdxOffset := IdxOffset + SIS_6_0.POSITION_STRINGLENGTH;
// Copy
MEMCPY(destAddr := ADR(TDQ.TU_ID), srcAddr := ADR(RecvTelegram[IdxOffset]), n := INT_TO_UDINT(SIS_6_0.TU_ID_STRINGLENGTH));
// Adjust index
IdxOffset := IdxOffset + SIS_6_0.TU_ID_STRINGLENGTH;
// Copy
MEMCPY(destAddr := ADR(TDQ.AssignmentID), srcAddr := ADR(RecvTelegram[IdxOffset]), n := INT_TO_UDINT(SIS_6_0.ASSIGNMENT_ID_STRINGLENGTH));
// Adjust index
IdxOffset := IdxOffset + SIS_6_0.ASSIGNMENT_ID_STRINGLENGTH;
// Copy
MEMCPY(destAddr := ADR(TDQ.MsgSequence), srcAddr := ADR(RecvTelegram[IdxOffset]), n := INT_TO_UDINT(SIS_6_0.MSG_SEQUENCE_STRINGLENGTH));
// Adjust index
IdxOffset := IdxOffset + SIS_6_0.MSG_SEQUENCE_STRINGLENGTH;
// Copy
MEMCPY(destAddr := ADR(TDQ.CODE), srcAddr := ADR(RecvTelegram[IdxOffset]), n := INT_TO_UDINT(SIS_6_0.TDQ_CODE_STRINGLENGTH));


// Map to ITC
TDQ_ITC.Position := TDQ.Position;
TDQ_ITC.Code := STRING_TO_INT(TDQ.Code);
TDQ_ITC.MsgSequence := STRING_TO_INT(TDQ.MsgSequence);
TDQ_ITC.AssignmentID := STRING_TO_UDINT(TDQ.AssignmentID);
TDQ_ITC.TU_ID := TDQ.TU_ID;

// Forward to mirror channel
M_MirrorData(Data := ADR(RecvTelegram), DataLen := ReceivedLength);

// Forward message to ITC
NoError := fbITC_Manager.M_AddData(
			meChannelSrc := Settings.MFCS_Channel,
			mMsgType	 := E_ITC_MsgTypeConv.TASK_DELETE_REQUEST,
			mpData		 := ADR(TDQ_ITC),
			mLen		 := SIZEOF(TDQ_ITC));


// If forwarding was successful
IF NoError THEN
	// Message processed
	fbBaseDriver.M_ProcessedMsg();
	
ELSE	
	DebugMsg := 'TDQ - Could not be forwarded to ITC';
	fbDebugMsg.M_SendErrorMsg(DebugMsg);	
END_IF
END_ACTION

ACTION A_PutTTA:
(**************************************************************************************
 * 	NAME		A_PutTTA
 * 	FUNCTION	Process TTA
 **************************************************************************************)

// Clear data structure 
MEMSET(destAddr := ADR(TTA), fillByte := 0, n := SIZEOF(TTA));

// Copy the TTA data fields to the TTA data structure 
IdxOffset := SIS_6_0.APP_DATA_OFFSET + 1;
// Copy
MEMCPY(destAddr := ADR(TTA.Position), srcAddr := ADR(RecvTelegram[IdxOffset]), n := INT_TO_UDINT(SIS_6_0.POSITION_STRINGLENGTH));
// Adjust index
IdxOffset := IdxOffset + SIS_6_0.POSITION_STRINGLENGTH;
// Copy
MEMCPY(destAddr := ADR(TTA.TU_DataIndex), srcAddr := ADR(RecvTelegram[IdxOffset]), n := INT_TO_UDINT(SIS_6_0.TU_DATAINDEX_STRINGLENGTH));
// Adjust index
IdxOffset := IdxOffset + SIS_6_0.TU_DATAINDEX_STRINGLENGTH;
// Copy
MEMCPY(destAddr := ADR(TTA.MsgSequence), srcAddr := ADR(RecvTelegram[IdxOffset]), n := INT_TO_UDINT(SIS_6_0.MSG_SEQUENCE_STRINGLENGTH));
// Adjust index
IdxOffset := IdxOffset + SIS_6_0.MSG_SEQUENCE_STRINGLENGTH;
// Copy
MEMCPY(destAddr := ADR(TTA.TU_ID), srcAddr := ADR(RecvTelegram[IdxOffset]), n := INT_TO_UDINT(SIS_6_0.TU_ID_STRINGLENGTH));
// Adjust index
IdxOffset := IdxOffset + SIS_6_0.TU_ID_STRINGLENGTH;
// Copy
MEMCPY(destAddr := ADR(TTA.TU_Type), srcAddr := ADR(RecvTelegram[IdxOffset]), n := INT_TO_UDINT(SIS_6_0.TU_TYPE_STRINGLENGTH));
// Adjust index
IdxOffset := IdxOffset + SIS_6_0.TU_TYPE_STRINGLENGTH;
// Copy
MEMCPY(destAddr := ADR(TTA.AssignmentID), srcAddr := ADR(RecvTelegram[IdxOffset]), n := INT_TO_UDINT(SIS_6_0.ASSIGNMENT_ID_STRINGLENGTH));
// Adjust index
IdxOffset := IdxOffset + SIS_6_0.ASSIGNMENT_ID_STRINGLENGTH;
// Copy
MEMCPY(destAddr := ADR(TTA.Length), srcAddr := ADR(RecvTelegram[IdxOffset]), n := INT_TO_UDINT(SIS_6_0.DIMENSIONS));
// Adjust index
IdxOffset := IdxOffset + SIS_6_0.DIMENSIONS;
// Copy
MEMCPY(destAddr := ADR(TTA.Width), srcAddr := ADR(RecvTelegram[IdxOffset]), n := INT_TO_UDINT(SIS_6_0.DIMENSIONS));
// Adjust index
IdxOffset := IdxOffset + SIS_6_0.DIMENSIONS;
// Copy
MEMCPY(destAddr := ADR(TTA.Height), srcAddr := ADR(RecvTelegram[IdxOffset]), n := INT_TO_UDINT(SIS_6_0.DIMENSIONS));
// Adjust index
IdxOffset := IdxOffset + SIS_6_0.DIMENSIONS;
// Copy
MEMCPY(destAddr := ADR(TTA.Weight), srcAddr := ADR(RecvTelegram[IdxOffset]), n := INT_TO_UDINT(SIS_6_0.TTA_WEIGHT));
// Adjust index
IdxOffset := IdxOffset + SIS_6_0.TTA_WEIGHT;
// Copy
MEMCPY(destAddr := ADR(TTA.Orientation), srcAddr := ADR(RecvTelegram[IdxOffset]), n := INT_TO_UDINT(SIS_6_0.TTA_ORIENTATION));
// Adjust index
IdxOffset := IdxOffset + SIS_6_0.TTA_ORIENTATION;
// Copy
MEMCPY(destAddr := ADR(TTA.TU_Parameter), srcAddr := ADR(RecvTelegram[IdxOffset]), n := INT_TO_UDINT(SIS_6_0.TTA_TU_PARAMETER));
// Adjust index
IdxOffset := IdxOffset + SIS_6_0.TTA_TU_PARAMETER;
// Copy
MEMCPY(destAddr := ADR(TTA.IO_Data), srcAddr := ADR(RecvTelegram[IdxOffset]), n := INT_TO_UDINT(SIS_6_0.TTA_IO_DATA_STRINGLENGTH));
// Adjust index
IdxOffset := IdxOffset + SIS_6_0.TTA_IO_DATA_STRINGLENGTH;
// Copy
MEMCPY(destAddr := ADR(TTA.LowerLimit), srcAddr := ADR(RecvTelegram[IdxOffset]), n := INT_TO_UDINT(SIS_6_0.TTA_LOWER_LIMIT_STRINGLENGTH));
// Adjust index
IdxOffset := IdxOffset + SIS_6_0.TTA_LOWER_LIMIT_STRINGLENGTH;
// Copy
MEMCPY(destAddr := ADR(TTA.UpperLimit), srcAddr := ADR(RecvTelegram[IdxOffset]), n := INT_TO_UDINT(SIS_6_0.TTA_UPPER_LIMIT_STRINGLENGTH));
// Adjust index
IdxOffset := IdxOffset + SIS_6_0.TTA_UPPER_LIMIT_STRINGLENGTH;
// Copy
MEMCPY(destAddr := ADR(TTA.GroupInfo), srcAddr := ADR(RecvTelegram[IdxOffset]), n := INT_TO_UDINT(SIS_6_0.TTA_GROUPINFO_STRINGLENGTH));
// Adjust index
IdxOffset := IdxOffset + SIS_6_0.TTA_GROUPINFO_STRINGLENGTH;
// Copy
MEMCPY(destAddr := ADR(TTA.Sequence), srcAddr := ADR(RecvTelegram[IdxOffset]), n := INT_TO_UDINT(SIS_6_0.TTA_SEQUENCE_STRINGLENGTH));
// Adjust index
IdxOffset := IdxOffset + SIS_6_0.TTA_SEQUENCE_STRINGLENGTH;
// Copy
MEMCPY(destAddr := ADR(TTA.NumberInSequence), srcAddr := ADR(RecvTelegram[IdxOffset]), n := INT_TO_UDINT(SIS_6_0.TTA_NO_IN_SEQUENCE_STRINGLENGTH));
// Adjust index
IdxOffset := IdxOffset + SIS_6_0.TTA_NO_IN_SEQUENCE_STRINGLENGTH;
// Copy
MEMCPY(destAddr := ADR(TTA.NumberOfDestinations), srcAddr := ADR(RecvTelegram[IdxOffset]), n := INT_TO_UDINT(SIS_6_0.TTA_NO_OF_DESTINATIONS_STRINGLENGTH));
// Adjust index
IdxOffset := IdxOffset + SIS_6_0.TTA_NO_OF_DESTINATIONS_STRINGLENGTH;

// Based on the "NumberOfDestinations in the TTA, obtain and store all the destinations 
FOR Idx := 1 TO STRING_TO_INT(TTA.NumberOfDestinations) DO
	// offset = ((Index - 1) * DestinationFieldLength  + BaseAddress ) 
	TempInt 		:= (((Idx - 1) * SIS_6_0.POSITION_STRINGLENGTH) + IdxOffset);
	MEMCPY(destAddr := ADR(TTA.Destination[idx]), srcAddr := ADR(RecvTelegram[TempInt]), n := INT_TO_UDINT(SIS_6_0.POSITION_STRINGLENGTH));
END_FOR

// Map to ITC
TTA_ITC.Position :=  TTA.Position;
TTA_ITC.TU_DataIndex := STRING_TO_INT(TTA.TU_DataIndex);
TTA_ITC.MsgSequence := STRING_TO_INT(TTA.MsgSequence);
TTA_ITC.TU_ID := TTA.TU_ID;
TTA_ITC.TU_Type := STRING_TO_INT(TTA.TU_Type);
TTA_ITC.AssignmentID := STRING_TO_UDINT(TTA.AssignmentID);
TTA_ITC.Length := STRING_TO_INT(TTA.Length);
TTA_ITC.Width := STRING_TO_INT(TTA.Width);
TTA_ITC.Height := STRING_TO_INT(TTA.Height);
TTA_ITC.Weight := STRING_TO_DINT(TTA.Weight);
TTA_ITC.Orientation := TTA.Orientation;
TTA_ITC.TU_Parameter := STRING_TO_INT(TTA.TU_Parameter);
TTA_ITC.IO_Data := STRING_TO_INT(TTA.IO_Data);
TTA_ITC.LowerLimit := STRING_TO_DINT(TTA.LowerLimit);
TTA_ITC.UpperLimit := STRING_TO_DINT(TTA.UpperLimit);
TTA_ITC.GroupID := STRING_TO_ULINT(TTA.GroupInfo);
TTA_ITC.Sequence := STRING_TO_ULINT(TTA.Sequence);
TTA_ITC.SubSequence := STRING_TO_INT(TTA.NumberInSequence);
TTA_ITC.NumberOfDestinations := STRING_TO_INT(TTA.NumberOfDestinations);
TTA_ITC.Destination := TTA.Destination;

// Forward to mirror channel
M_MirrorData(Data := ADR(RecvTelegram), DataLen := ReceivedLength);

// Forward message to ITC
NoError := fbITC_Manager.M_AddData(
			meChannelSrc := Settings.MFCS_Channel,
			mMsgType	 := E_ITC_MsgTypeConv.TRANSPORT_TASK_ASSIGNMENT,
			mpData		 := ADR(TTA_ITC),
			mLen		 := SIZEOF(TTA_ITC));

// If forwarding was successful
IF NoError THEN
	// Message processed
	fbBaseDriver.M_ProcessedMsg();
ELSE	
	DebugMsg := 'TTA - Could not be forwarded to ITC';
	fbDebugMsg.M_SendErrorMsg(DebugMsg);	
END_IF
END_ACTION

ACTION A_PutTUQ:
(**************************************************************************************
 * 	NAME		A_PutTUQ
 * 	FUNCTION	Process TUQ
 **************************************************************************************)

// Clear data structure 
MEMSET(destAddr := ADR(TUQ), fillByte := 0, n := SIZEOF(TUQ));

// Copy the TUQ data fields to the TUQ data structure 
IdxOffset := SIS_6_0.APP_DATA_OFFSET + 1;

MEMCPY(destAddr := ADR(TUQ.TU_ID), srcAddr := ADR(RecvTelegram[IdxOffset]), n := INT_TO_UDINT(SIS_6_0.TU_ID_STRINGLENGTH));

// Adjust index
IdxOffset := IdxOffset + SIS_6_0.TU_ID_STRINGLENGTH;

MEMCPY(destAddr := ADR(TUQ.AssignmentID), srcAddr := ADR(RecvTelegram[IdxOffset]), n := INT_TO_UDINT(SIS_6_0.ASSIGNMENT_ID_STRINGLENGTH));

// Map to ITC
TUQ_ITC.AssignmentID := STRING_TO_UDINT(TUQ.AssignmentID);
TUQ_ITC.TU_ID := TUQ.TU_ID;

// Forward to mirror channel
M_MirrorData(Data := ADR(RecvTelegram), DataLen := ReceivedLength);

// Forward message to ITC
NoError := fbITC_Manager.M_AddData(
			meChannelSrc := Settings.MFCS_Channel,
			mMsgType	 := E_ITC_MsgTypeConv.TRANSPORT_UNIT_REQUEST,
			mpData		 := ADR(TUQ_ITC),
			mLen		 := SIZEOF(TUQ_ITC));
				
// If forwarding was successful
IF NoError THEN
	// Message processed
	fbBaseDriver.M_ProcessedMsg();
	
ELSE	
	DebugMsg := 'TUQ - Could not be forwarded to ITC';
	fbDebugMsg.M_SendErrorMsg(DebugMsg);	
END_IF
END_ACTION

ACTION A_PutVIQ:
(**************************************************************************************
 * 	NAME		A_PutVIQ
 * 	FUNCTION	Process VIQ
 **************************************************************************************)
 
// Clear data structure 
MEMSET(destAddr := ADR(VIQ), fillByte := 0, n := SIZEOF(VIQ));

// Copy the VIQ data fields to the VIQ data structure 
IdxOffset := SIS_6_0.APP_DATA_OFFSET + 1;
// Copy
MEMCPY(destAddr := ADR(VIQ.Position), srcAddr := ADR(RecvTelegram[IdxOffset]), n := INT_TO_UDINT(SIS_6_0.POSITION_STRINGLENGTH));
// Adjust index
IdxOffset := IdxOffset + SIS_6_0.POSITION_STRINGLENGTH;
//Copy
MEMCPY(destAddr := ADR(VIQ.NumberOfKeys), srcAddr := ADR(RecvTelegram[IdxOffset]), n := INT_TO_UDINT(SIS_6_0.VIQ_NUMBER_OF_KEYS_STRINGLENGTH));
// Adjust index
IdxOffset := IdxOffset + SIS_6_0.VIQ_NUMBER_OF_KEYS_STRINGLENGTH;

IF STRING_TO_INT(VIQ.NumberOfKeys) <= System.NUMBER_OF_KEYS_VIQ THEN
	FOR Idx := 1 TO STRING_TO_INT(VIQ.NumberOfKeys) BY 1 DO
		// Copy
		MEMCPY(destAddr := ADR(VIQ.Keys[Idx]), srcAddr := ADR(RecvTelegram[IdxOffset]), n := INT_TO_UDINT(SIS_6_0.VIQ_KEY_STRINGLENGTH));
		// Adjust index
		IdxOffset := IdxOffset + SIS_6_0.VIQ_KEY_STRINGLENGTH; 
	END_FOR
END_IF
// Map to ITC
VIQ_ITC.Position := VIQ.Position;
VIQ_ITC.NumberOfKeys := STRING_TO_INT(VIQ.NumberOfKeys);
VIQ_ITC.Keys := VIQ.Keys;

// Forward to mirror channel
M_MirrorData(Data := ADR(RecvTelegram), DataLen := ReceivedLength);

// Forward message to ITC
NoError := fbITC_Manager.M_AddData(
			meChannelSrc := Settings.MFCS_Channel,
			mMsgType	 := E_ITC_MsgTypeConv.VISUALIZATION_INFORMATION_REQUEST,
			mpData		 := ADR(VIQ_ITC),
			mLen		 := SIZEOF(VIQ_ITC));

// If forwarding was successful
IF NoError THEN
	// Message processed
	fbBaseDriver.M_ProcessedMsg();
	
ELSE	
	DebugMsg := 'VIQ - Could not be forwarded to ITC';
	fbDebugMsg.M_SendErrorMsg(DebugMsg);	
END_IF
END_ACTION

METHOD M_BufferLevelAlarm : BOOL
(**************************************************************************************
 * 	Application		:	BoxControl Framework
 *	Revision		:	$Revision: 404529 $
 *	Revision date	:	$Date: 2018-04-23 08:21:38 +0200 (Mo., 23 Apr 2018) $
 *	Last changed by	:	$Author: b7bolm $
 *	URL				:	$URL: http://almscdc.swisslog.com/repo/SWPD/Development/BoxControlFramework/20_Release/trunk/01_Software/BCF/BCF/JumpStart/20_Product/10_App/11_Com/10_Lib/10_Conv/12_MFCS/11_SIS/FB_SIS_MsgManager_6_0.TcPOU $
 *
 *	Purpose			:	If buffer fill quantity exeeds a certain level, return an
 *						alarm.
 *
 * ------------------------------------------------------------------------------------
 *	Copyright Swisslog [IP AG], Switzerland. All rights reserved.
 * 
 * ------------------------------------------------------------------------------------
 *	
 * 	Revision History: 
 *
 * 	VERSION			DATE			INITIALS			DESCRIPTION
 *	0.1				01.01.2001		swl					Example
 *
 **************************************************************************************)
// Set bufffer alarm if buffer level exeeds a certain level
IF fbBaseDriver.SendBufferQuantity > Settings.BufferLevelAlarm THEN
	BufferAlarmActive := TRUE;
	
// Reset bufffer alarm if buffer level is lower the hyst	
ELSIF BufferAlarmActive AND
	  fbBaseDriver.SendBufferQuantity < Settings.BufferLevelAlarm - Settings.BufferLevelHysterese THEN
	BufferAlarmActive := FALSE;
END_IF

M_BufferLevelAlarm := BufferAlarmActive;
END_METHOD

METHOD M_BufferLevelWarning : BOOL
(**************************************************************************************
 * 	Application		:	BoxControl Framework
 *	Revision		:	$Revision: 404529 $
 *	Revision date	:	$Date: 2018-04-23 08:21:38 +0200 (Mo., 23 Apr 2018) $
 *	Last changed by	:	$Author: b7bolm $
 *	URL				:	$URL: http://almscdc.swisslog.com/repo/SWPD/Development/BoxControlFramework/20_Release/trunk/01_Software/BCF/BCF/JumpStart/20_Product/10_App/11_Com/10_Lib/10_Conv/12_MFCS/11_SIS/FB_SIS_MsgManager_6_0.TcPOU $
 *
 *	Purpose			:	If buffer fill quantity exeeds a certain level, return a
 *						warning.
 *
 * ------------------------------------------------------------------------------------
 *	Copyright Swisslog [IP AG], Switzerland. All rights reserved.
 * 
 * ------------------------------------------------------------------------------------
 *	
 * 	Revision History: 
 *
 * 	VERSION			DATE			INITIALS			DESCRIPTION
 *	0.1				01.01.2001		swl					Example
 *
 **************************************************************************************)
// Set buffer warning if buffer level exeeds a certain level
IF fbBaseDriver.SendBufferQuantity > Settings.BufferLevelWarning THEN
	BufferWarningActive := TRUE;
	
// Reset buffer warning if buffer level is lower the hyst	
ELSIF BufferWarningActive AND
	  fbBaseDriver.SendBufferQuantity < Settings.BufferLevelWarning - Settings.BufferLevelHysterese THEN
	BufferWarningActive := FALSE;
END_IF

M_BufferLevelWarning := BufferWarningActive;
END_METHOD

{attribute 'object_name' := 'M_CallCommunicationService'}
METHOD M_CallCommunicationService
(**************************************************************************************
 * 	Application		:	BoxControl Framework
 *	Revision		:	$Revision: 404529 $
 *	Revision date	:	$Date: 2018-04-23 08:21:38 +0200 (Mo., 23 Apr 2018) $
 *	Last changed by	:	$Author: b7bolm $
 *	URL				:	$URL: http://almscdc.swisslog.com/repo/SWPD/Development/BoxControlFramework/20_Release/trunk/01_Software/BCF/BCF/JumpStart/20_Product/10_App/11_Com/10_Lib/10_Conv/12_MFCS/11_SIS/FB_SIS_MsgManager_6_0.TcPOU $
 *
 *	Purpose			:	Call communication service
 *
 * ------------------------------------------------------------------------------------
 *	Copyright Swisslog [IP AG], Switzerland. All rights reserved.
 * 
 * ------------------------------------------------------------------------------------
 *	
 * 	Revision History: 
 *
 * 	VERSION			DATE			INITIALS			DESCRIPTION
 *	0.1				01.01.2001		swl					Example
 *
 **************************************************************************************)

(**************************************************************************************************************
 	Initialization
***************************************************************************************************************)
M_Init(FALSE);


(**************************************************************************************************************
   Call SIS BaseDriver
***************************************************************************************************************)
fbBaseDriver(
	Settings 		   := Settings.BaseDriver,
	pRecvAppData	   := ADR(RecvTelegram),
	RecvAppDataLen	   := SIZEOF(RecvTelegram),
	ReceivedAppDataLen => ReceivedLength);


(**************************************************************************************************************
   Buffering incoming data 
***************************************************************************************************************)
(*
It is possible, that the currently processed telegram, takes longer 
than one cycle. Therefore by the base driver provided data needs to 
be buffered.
*)

// If new application data are available
IF fbBaseDriver.NewAppData THEN
	// Get the TYPE of telegram which was received 
	MEMCPY(destAddr := ADR(TelegramType), srcAddr := ADR(RecvTelegram), n := 3);
	
	// Transport Task Assignment
	IF TelegramType = 'TTA' THEN
		// Process
		A_PutTTA();
		
	// Transport Delete Request
	ELSIF TelegramType = 'TDQ' THEN
		// Process
		A_PutTDQ();
	
	// Subsystem Control Request
	ELSIF TelegramType = 'SCQ' THEN	
		// Process
		A_PutSCQ();
	
	// Group Control Request
	ELSIF TelegramType = 'RAA' THEN
		// Process
		A_PutRAA();
	
	// Visualisation Information Request
	ELSIF TelegramType = 'VIQ' THEN
		// Process
		A_PutVIQ();	
	
	// Robot Delete Request		
	ELSIF TelegramType = 'RDQ' THEN
		// Process
		A_PutRDQ();
	
	// Group Control Request
	ELSIF TelegramType = 'GCQ' THEN	
		// Process
		A_PutGCQ();
	
	// Element Control Request
	ELSIF TelegramType = 'ECQ' THEN	
		// Process
		A_PutECQ();
	
	// Function Control Request
	ELSIF TelegramType = 'FCQ' THEN	
		// Process
		A_PutFCQ();
	
	// Subsystem Status Request
	ELSIF TelegramType = 'SSQ' THEN	
		// Process
		A_PutSSQ();
	
	// Group Status Request
	ELSIF TelegramType = 'GSQ' THEN	
		// Process
		A_PutGSQ();
		
	// Element Status Request
	ELSIF TelegramType = 'ESQ' THEN	
		// Process
		A_PutESQ();
	
	// Function Status Request
	ELSIF TelegramType = 'FSQ' THEN	
		// Process
		A_PutFSQ();

	// Transport Unit Request
	ELSIF TelegramType = 'TUQ' THEN	
		// Process
		A_PutTUQ();
	
	// Scanner Information Request
	ELSIF TelegramType = 'SIQ' THEN	
		// Process
		A_PutSIQ();

	// Manual Control Request
	ELSIF TelegramType = 'MCQ' THEN	
		// Process
		A_PutMCQ();
	
	// Digital Input Request
	ELSIF TelegramType = 'DIQ' THEN	
		// Process
		A_PutDIQ();
	
	// Set Digital Output
	ELSIF TelegramType = 'SDO' THEN	
		// Process
		A_PutSDO();
		
	// I/O Status Request
	ELSIF TelegramType = 'IRQ' THEN	
		// Process
		A_PutIRQ();
	
	// Global Variable Request
	ELSIF TelegramType = 'GVQ' THEN	
		// Process
		A_PutGVQ();
		
	// Customized message
	ELSIF TelegramType = 'MSG' THEN	
		// Process
		M_PutMSG(ADR(RecvTelegram),ReceivedLength);
			
	// Data Aquisition Request
	ELSIF TelegramType = 'DAQ' THEN	
		// Process
		A_PutDAQ();
		
	// Gathered Data Request
	ELSIF TelegramType = 'GDQ' THEN	
		// Process
		A_PutGDQ();		
	// Drop unknown types
	ELSE
		// Message processed
		fbBaseDriver.M_ProcessedMsg();
	END_IF
ELSE
	// Clear received structure
	MEMSET(destAddr := ADR(RecvTelegram), fillByte := 0, n := SIZEOF(RecvTelegram));
END_IF
END_METHOD

METHOD M_GetReceivedData : ST_PointerSet
(**************************************************************************************
 * 	Application		:	BoxControl Framework
 *	Revision		:	$Revision: 404529 $
 *	Revision date	:	$Date: 2018-04-23 08:21:38 +0200 (Mo., 23 Apr 2018) $
 *	Last changed by	:	$Author: b7bolm $
 *	URL				:	$URL: http://almscdc.swisslog.com/repo/SWPD/Development/BoxControlFramework/20_Release/trunk/01_Software/BCF/BCF/JumpStart/20_Product/10_App/11_Com/10_Lib/10_Conv/12_MFCS/11_SIS/FB_SIS_MsgManager_6_0.TcPOU $
 *
 *	Purpose			:	Returns last received data
 *
 * ------------------------------------------------------------------------------------
 *	Copyright Swisslog [IP AG], Switzerland. All rights reserved.
 * 
 * ------------------------------------------------------------------------------------
 *	
 * 	Revision History: 
 *
 * 	VERSION			DATE			INITIALS			DESCRIPTION
 *	0.1				01.01.2001		swl					Example
 *
 **************************************************************************************)

M_GetReceivedData.pAdr := ADR(RecvTelegram);
M_GetReceivedData.Len := ReceivedLength;
END_METHOD

METHOD M_Init : BOOL
(**************************************************************************************
 * 	Application		:	BoxControl Framework
 *	Revision		:	$Revision: 404529 $
 *	Revision date	:	$Date: 2018-04-23 08:21:38 +0200 (Mo., 23 Apr 2018) $
 *	Last changed by	:	$Author: b7bolm $
 *	URL				:	$URL: http://almscdc.swisslog.com/repo/SWPD/Development/BoxControlFramework/20_Release/trunk/01_Software/BCF/BCF/JumpStart/20_Product/10_App/11_Com/10_Lib/10_Conv/12_MFCS/11_SIS/FB_SIS_MsgManager_6_0.TcPOU $
 *
 *	Purpose			:	Initialize Msg Manager.
 *
 * ------------------------------------------------------------------------------------
 *	Copyright Swisslog [IP AG], Switzerland. All rights reserved.
 * 
 * ------------------------------------------------------------------------------------
 *	
 * 	Revision History: 
 *
 * 	VERSION			DATE			INITIALS			DESCRIPTION
 *	0.1				01.01.2001		swl					Example
 *
 **************************************************************************************)
VAR_INPUT
	mInit		: BOOL; // Force init
END_VAR
// If instance is not initialized or init is forced
IF NOT Init OR mInit THEN
	
	// Activate configuration
	Settings := Config;
	fbBaseDriver.Settings := Settings.BaseDriver;
	
	// Initialize base driver
	fbBaseDriver.M_Init(TRUE);

    // Send log message
    fbDebugMsg.M_SendInfoMsg('Initialization done');
		
	// Init done
    Init := TRUE;

END_IF
END_METHOD

{attribute 'object_name' := 'M_IsConnected'}
METHOD M_IsConnected : BOOL
(**************************************************************************************
 * 	Application		:	BoxControl Framework
 *	Revision		:	$Revision: 404529 $
 *	Revision date	:	$Date: 2018-04-23 08:21:38 +0200 (Mo., 23 Apr 2018) $
 *	Last changed by	:	$Author: b7bolm $
 *	URL				:	$URL: http://almscdc.swisslog.com/repo/SWPD/Development/BoxControlFramework/20_Release/trunk/01_Software/BCF/BCF/JumpStart/20_Product/10_App/11_Com/10_Lib/10_Conv/12_MFCS/11_SIS/FB_SIS_MsgManager_6_0.TcPOU $
 *
 *	Purpose			:	Connection is established
 *
 * ------------------------------------------------------------------------------------
 *	Copyright Swisslog [IP AG], Switzerland. All rights reserved.
 * 
 * ------------------------------------------------------------------------------------
 *	
 * 	Revision History: 
 *
 * 	VERSION			DATE			INITIALS			DESCRIPTION
 *	0.1				01.01.2001		swl					Example
 *
 **************************************************************************************)

// Return connection state of base driver
M_IsConnected := fbBaseDriver.Connected;
END_METHOD

METHOD PROTECTED M_MirrorData : BOOL
(**************************************************************************************
 * 	Application		:	BoxControl Framework
 *	Revision		:	$Revision: 404529 $
 *	Revision date	:	$Date: 2018-04-23 08:21:38 +0200 (Mo., 23 Apr 2018) $
 *	Last changed by	:	$Author: b7bolm $
 *	URL				:	$URL: http://almscdc.swisslog.com/repo/SWPD/Development/BoxControlFramework/20_Release/trunk/01_Software/BCF/BCF/JumpStart/20_Product/10_App/11_Com/10_Lib/10_Conv/12_MFCS/11_SIS/FB_SIS_MsgManager_6_0.TcPOU $
 *
 *	Purpose			:	Mirror these data (Max length 255) to a additonal connection.
 *
 * ------------------------------------------------------------------------------------
 *	Copyright Swisslog [IP AG], Switzerland. All rights reserved.
 * 
 * ------------------------------------------------------------------------------------
 *	
 * 	Revision History: 
 *
 * 	VERSION			DATE			INITIALS			DESCRIPTION
 *	0.1				01.01.2001		swl					Example
 *
 **************************************************************************************)
VAR_INPUT
	Data	: PVOID;
	DataLen	: UDINT;
END_VAR
// Initialize
M_MirrorData := TRUE;

// Check if a mirror channel is available
IF Settings.MirrorChannel > E_MFCS_Channel.BEGIN_CHANNEL AND
   Settings.MirrorChannel < E_MFCS_Channel.END_CHANNEL THEN
   
   	// Forward data to an additional connection
   	M_MirrorData := fbMFCS_Channel[Settings.MirrorChannel].M_SendData(
						meChannelSrc := 0,
						mMsgType  	 := E_ITC_MsgTypeConv.DATA_MESSAGE,
						mpData	  	 := Data,
						mLen		 := DataLen);
				
   	// If forwarding was not successful
   	IF NOT M_MirrorData THEN
		DebugMsg := 'Mirror Channel was not able to accept message.';
		fbDebugMsg.M_SendErrorMsg(DebugMsg);		
   	END_IF
END_IF
END_METHOD

METHOD PROTECTED M_ProcessATR : BOOL
(**************************************************************************************
 * 	Application		:	BoxControl Framework
 *	Revision		:	$Revision: 404529 $
 *	Revision date	:	$Date: 2018-04-23 08:21:38 +0200 (Mo., 23 Apr 2018) $
 *	Last changed by	:	$Author: b7bolm $
 *	URL				:	$URL: http://almscdc.swisslog.com/repo/SWPD/Development/BoxControlFramework/20_Release/trunk/01_Software/BCF/BCF/JumpStart/20_Product/10_App/11_Com/10_Lib/10_Conv/12_MFCS/11_SIS/FB_SIS_MsgManager_6_0.TcPOU $
 *
 *	Purpose			:	Send ATR
 *
 * ------------------------------------------------------------------------------------
 *	Copyright Swisslog [IP AG], Switzerland. All rights reserved.
 * 
 * ------------------------------------------------------------------------------------
 *	
 * 	Revision History: 
 *
 * 	VERSION			DATE			INITIALS			DESCRIPTION
 *	0.1				01.01.2001		swl					Example
 *
 **************************************************************************************)
VAR_INPUT
 	meChannelSrc		: E_MFCS_Channel; // Source communicaton channel
	mpATR				: POINTER TO ST_ITC_ATR; // Pointer to ATR
END_VAR
(**************************************************************************************************************
 	Check if a telegram needs to be send
***************************************************************************************************************)
// If settings allow sending a ATR 	
IF  Settings.Telegrams.SendATR THEN
	// If the source of the request is this channel or is undefined
	IF meChannelSrc = Settings.MFCS_Channel OR
		meChannelSrc = E_MFCS_Channel.BEGIN_CHANNEL THEN
		;//Proceed
	ELSE // Source is a different MFCS Connection
		// Dont send a telegram		
		RETURN;
	END_IF	
ELSE
	// Dont send a telegram		
	RETURN;
END_IF

(**************************************************************************************************************
 	ITC - Map generic data to type
***************************************************************************************************************)
MEMCPY(destAddr := ADR(ATR_ITC), srcAddr := mpATR, n := SIZEOF(ATR_ITC));

(**************************************************************************************************************
 	Formatting data
***************************************************************************************************************)
// Fill position
ATR.Position	:= 	F_StuffString(
						InputString 	:= ATR_ITC.Position, 
						StringLength	:= SIS_6_0.POSITION_STRINGLENGTH, 
						StuffCharacter 	:= '0',
						LeftAligned		:= FALSE);

// Get Error Code 
ATR.ReturnCode := F_StuffString(
					InputString 	:= INT_TO_STRING(ATR_ITC.ReturnCode), 
					StringLength	:= SIS_6_0.ERRORCODE_STRINGLENGTH, 
					StuffCharacter 	:= '0',
					LeftAligned		:= FALSE);
					
(**************************************************************************************************************
 	Build byte stream and add to Base Driver
***************************************************************************************************************)
// Initialize
MEMSET(destAddr := ADR(SendTelegram), 0, SIZEOF(SendTelegram));
WritePointer := 0;

F_AssembleByteStream(
	pSrc:= ADR('ATR'), 
	SrcLen:= 3, 
	pDest:= ADR(SendTelegram), 
	DestLen:= SIZEOF(SendTelegram), 
	WritePointer:= WritePointer);

F_AssembleByteStream(
	pSrc:= ADR(ATR.Position), 
	SrcLen:= INT_TO_UDINT(LEN(ATR.Position)), 
	pDest:= ADR(SendTelegram), 
	DestLen:= SIZEOF(SendTelegram), 
	WritePointer:= WritePointer);

F_AssembleByteStream(
	pSrc:= ADR(ATR.ReturnCode), 
	SrcLen:= INT_TO_UDINT(LEN(ATR.ReturnCode)), 
	pDest:= ADR(SendTelegram), 
	DestLen:= SIZEOF(SendTelegram), 
	WritePointer:= WritePointer);
	
// Add to buffer of Base Driver
M_ProcessATR := fbBaseDriver.M_SendAppData(
					mpSendData := ADR(SendTelegram),
					mSendDataLen := WritePointer);

// Forward to mirror channel
M_MirrorData(Data := ADR(SendTelegram), DataLen := WritePointer);
END_METHOD

METHOD PROTECTED M_ProcessDAR : BOOL
(**************************************************************************************
 * 	Application		:	BoxControl Framework
 *	Revision		:	$Revision: 404529 $
 *	Revision date	:	$Date: 2018-04-23 08:21:38 +0200 (Mo., 23 Apr 2018) $
 *	Last changed by	:	$Author: b7bolm $
 *	URL				:	$URL: http://almscdc.swisslog.com/repo/SWPD/Development/BoxControlFramework/20_Release/trunk/01_Software/BCF/BCF/JumpStart/20_Product/10_App/11_Com/10_Lib/10_Conv/12_MFCS/11_SIS/FB_SIS_MsgManager_6_0.TcPOU $
 *
 *	Purpose			:	Send DAR
 *
 * ------------------------------------------------------------------------------------
 *	Copyright Swisslog [IP AG], Switzerland. All rights reserved.
 * 
 * ------------------------------------------------------------------------------------
 *	
 * 	Revision History: 
 *
 * 	VERSION			DATE			INITIALS			DESCRIPTION
 *	0.1				01.01.2001		swl					Example
 *
 **************************************************************************************)
VAR_INPUT
 	meChannelSrc		: E_MFCS_Channel; // Source communicaton channel
	mpDAR				: POINTER TO ST_ITC_DAR; // Pointer to DAR
END_VAR
VAR
	Idx : INT;	//Iterator
	Idx2 : INT;	//Iterator
END_VAR
(**************************************************************************************************************
 	Check if a telegram needs to be send
***************************************************************************************************************)
// If settings allow sending a DAR 	
IF  Settings.Telegrams.SendDAR THEN
	// If the source of the request is this channel or is undefined
	IF meChannelSrc = Settings.MFCS_Channel OR
		meChannelSrc = E_MFCS_Channel.BEGIN_CHANNEL THEN
		;//Proceed
	ELSE // Source is a different MFCS Connection
		// Dont send a telegram		
		RETURN;
	END_IF	
ELSE
	// Dont send a telegram		
	RETURN;
END_IF

(**************************************************************************************************************
 	ITC - Map generic data to type
***************************************************************************************************************)
MEMCPY(destAddr := ADR(DAR_ITC), srcAddr := mpDAR, n := SIZEOF(DAR_ITC));
MEMSET(destAddr := ADR(DAR), 0, SIZEOF(DAR));
(**************************************************************************************************************
 	Formatting data
***************************************************************************************************************)


// Get SIS-Number 
DAR.Position := F_StuffString(
					InputString 	:= DAR_ITC.Position, 
					StringLength	:= SIS_6_0.POSITION_STRINGLENGTH, 
					StuffCharacter 	:= '0', 
					LeftAligned := FALSE);
//Get Number Sets
DAR.NumberOfSets := F_StuffString(
						InputString 	:= INT_TO_STRING(DAR_ITC.NumberOfSets), 
						StringLength	:= SIS_6_0.DATA_ACQUISITION_NUMBEROFSETS, 
						StuffCharacter 	:= '0', 
						LeftAligned := FALSE);
//Get  Code
DAR.Code := F_StuffString(
						InputString 	:= INT_TO_STRING(DAR_ITC.Code), 
						StringLength	:= SIS_6_0.DATA_ACQUISITION_CODE, 
						StuffCharacter 	:= '0', 
						LeftAligned 	:= FALSE);

//Build Set 
IF DAR_ITC.SetOffset>E_CM_Index.E_BEGIN_VARIABLE THEN 	
Idx2:=1;	
	FOR Idx:=DAR_ITC.SetOffset TO DAR_ITC.NumberOfSets+DAR_ITC.SetOffset -1  DO 
		DAR.Set[Idx2]   := CONCAT(DAR.Set[Idx2],F_StuffString(InputString :=DAR_ITC.Set[Idx].mVariableName, StringLength:= System.CM_VARIABLENAME_STRINGLENGTH, StuffCharacter:= ' ', LeftAligned := FALSE));
		DAR.Set[Idx2]   := CONCAT(DAR.Set[Idx2],F_Time_TO_MaxReportTime(TIN:= DAR_ITC.Set[Idx].MaxReportTime));
		DAR.Set[Idx2]   := CONCAT(DAR.Set[Idx2],F_Time_TO_SampleTime(DAR_ITC.Set[Idx].SampleTime));
		DAR.Set[Idx2]   := CONCAT(DAR.Set[Idx2],F_StuffString(InputString := INT_TO_STRING(DAR_ITC.Set[Idx].Threshold), StringLength:= SIS_6_0.DATA_ACQUISITION_THRESHOLD, StuffCharacter:= '0', LeftAligned := FALSE));
		DAR.Set[Idx2]   := CONCAT(DAR.Set[Idx2],F_StuffString(InputString := INT_TO_STRING(BOOL_TO_INT(DAR_ITC.Set[Idx].Option)), StringLength:= 1, StuffCharacter:= '0', LeftAligned := FALSE));
		DAR.Set[Idx2]   := CONCAT(DAR.Set[Idx2],F_StuffString(InputString := INT_TO_STRING(BOOL_TO_INT(DAR_ITC.Set[Idx].Enable)), StringLength:= 1, StuffCharacter:= '0', LeftAligned := FALSE));
		DAR.Set[Idx2]   := CONCAT(DAR.Set[Idx2],F_StuffString(InputString := INT_TO_STRING(DAR_ITC.Set[Idx].ErrorCode), StringLength:= 4, StuffCharacter:= '0', LeftAligned := FALSE));
		Idx2:= Idx2+1;
	END_FOR
ELSE  	
	FOR Idx:=1 TO DAR_ITC.NumberOfSets DO 
		DAR.Set[Idx]   := CONCAT(DAR.Set[Idx],F_StuffString(InputString :=DAR_ITC.Set[Idx].mVariableName, StringLength:= System.CM_VARIABLENAME_STRINGLENGTH, StuffCharacter:= ' ', LeftAligned := FALSE));
		DAR.Set[Idx]   := CONCAT(DAR.Set[Idx],F_Time_TO_MaxReportTime(TIN:= DAR_ITC.Set[Idx].MaxReportTime));
		DAR.Set[Idx]   := CONCAT(DAR.Set[Idx],F_Time_TO_SampleTime(DAR_ITC.Set[Idx].SampleTime));
		DAR.Set[Idx]   := CONCAT(DAR.Set[Idx],F_StuffString(InputString := INT_TO_STRING(DAR_ITC.Set[Idx].Threshold), StringLength:= SIS_6_0.DATA_ACQUISITION_THRESHOLD, StuffCharacter:= '0', LeftAligned := FALSE));
		DAR.Set[Idx]   := CONCAT(DAR.Set[Idx],F_StuffString(InputString := INT_TO_STRING(BOOL_TO_INT(DAR_ITC.Set[Idx].Option)), StringLength:= 1, StuffCharacter:= '0', LeftAligned := FALSE));
		DAR.Set[Idx]   := CONCAT(DAR.Set[Idx],F_StuffString(InputString := INT_TO_STRING(BOOL_TO_INT(DAR_ITC.Set[Idx].Enable)), StringLength:= 1, StuffCharacter:= '0', LeftAligned := FALSE));
		DAR.Set[Idx]   := CONCAT(DAR.Set[Idx],F_StuffString(InputString := INT_TO_STRING(DAR_ITC.Set[Idx].ErrorCode), StringLength:= 4, StuffCharacter:= '0', LeftAligned := FALSE));
	END_FOR
END_IF;
	

(**************************************************************************************************************
 Build string and add to Base Driver
***************************************************************************************************************)
MEMSET(destAddr := ADR(SendTelegram), 0, SIZEOF(SendTelegram));
WritePointer := 0;

F_AssembleByteStream(
	pSrc:= ADR('DAR'), 
	SrcLen:= 3, 
	pDest:= ADR(SendTelegram), 
	DestLen:= SIZEOF(SendTelegram), 
	WritePointer:= WritePointer);

F_AssembleByteStream(
	pSrc:= ADR(DAR.Position), 
	SrcLen:= INT_TO_UDINT(LEN(DAR.Position)), 
	pDest:= ADR(SendTelegram), 
	DestLen:= SIZEOF(SendTelegram), 
	WritePointer:= WritePointer);

F_AssembleByteStream(
	pSrc:= ADR(DAR.Code), 
	SrcLen:= INT_TO_UDINT(LEN(DAR.Code)), 
	pDest:= ADR(SendTelegram), 
	DestLen:= SIZEOF(SendTelegram), 
	WritePointer:= WritePointer);
	
F_AssembleByteStream(
	pSrc:= ADR(DAR.NumberOfSets), 
	SrcLen:= INT_TO_UDINT(LEN(DAR.NumberOfSets)), 
	pDest:= ADR(SendTelegram), 
	DestLen:= SIZEOF(SendTelegram), 
	WritePointer:= WritePointer);
	
IF DAR_ITC.SetOffset>E_CM_Index.E_BEGIN_VARIABLE THEN 	
Idx2:=1;	
	FOR Idx:=DAR_ITC.SetOffset TO DAR_ITC.NumberOfSets+DAR_ITC.SetOffset -1  DO 
		F_AssembleByteStream(
						pSrc			:= ADR(DAR.Set[Idx2]), 
						SrcLen			:= INT_TO_UDINT(LEN(DAR.Set[Idx2])), 
						pDest			:= ADR(SendTelegram), 
						DestLen			:= SIZEOF(SendTelegram), 
						WritePointer	:= WritePointer);
		Idx2 := Idx2 +1;
	END_FOR;
ELSE
	FOR Idx:=1 TO DAR_ITC.NumberOfSets DO 
		F_AssembleByteStream(
						pSrc			:= ADR(DAR.Set[Idx]), 
						SrcLen			:= INT_TO_UDINT(LEN(DAR.Set[Idx])), 
						pDest			:= ADR(SendTelegram), 
						DestLen			:= SIZEOF(SendTelegram), 
						WritePointer	:= WritePointer);
	END_FOR;
END_IF
	

// Add to buffer of Base Driver
M_ProcessDAR := fbBaseDriver.M_SendAppData(
					mpSendData := ADR(SendTelegram),
					mSendDataLen := WritePointer);
					
// Forward to mirror channel
M_MirrorData(Data := ADR(SendTelegram), DataLen := WritePointer);
END_METHOD

METHOD PROTECTED M_ProcessECR : BOOL
(**************************************************************************************
 * 	Application		:	BoxControl Framework
 *	Revision		:	$Revision: 404529 $
 *	Revision date	:	$Date: 2018-04-23 08:21:38 +0200 (Mo., 23 Apr 2018) $
 *	Last changed by	:	$Author: b7bolm $
 *	URL				:	$URL: http://almscdc.swisslog.com/repo/SWPD/Development/BoxControlFramework/20_Release/trunk/01_Software/BCF/BCF/JumpStart/20_Product/10_App/11_Com/10_Lib/10_Conv/12_MFCS/11_SIS/FB_SIS_MsgManager_6_0.TcPOU $
 *
 *	Purpose			:	Send ECR
 *
 * ------------------------------------------------------------------------------------
 *	Copyright Swisslog [IP AG], Switzerland. All rights reserved.
 * 
 * ------------------------------------------------------------------------------------
 *	
 * 	Revision History: 
 *
 * 	VERSION			DATE			INITIALS			DESCRIPTION
 *	0.1				01.01.2001		swl					Example
 *
 **************************************************************************************)
 
VAR_INPUT
 	meChannelSrc		: E_MFCS_Channel; // Source communicaton channel
	mpECR				: POINTER TO ST_ITC_ECR; // Pointer to ECR
END_VAR
(**************************************************************************************************************
 	Check if a telegram needs to be send
***************************************************************************************************************)
// If settings allow sending a ECR 	
IF  Settings.Telegrams.SendECR THEN
	// If the source of the request is this channel or is undefined
	IF meChannelSrc = Settings.MFCS_Channel OR
		meChannelSrc = E_MFCS_Channel.BEGIN_CHANNEL THEN
		;//Proceed
	ELSE // Source is a different MFCS Connection
		// Dont send a telegram		
		RETURN;
	END_IF	
ELSE
	// Dont send a telegram		
	RETURN;
END_IF

(**************************************************************************************************************
 	ITC - Map generic data to type
***************************************************************************************************************)
MEMCPY(destAddr := ADR(ECR_ITC), srcAddr := mpECR, n := SIZEOF(ECR_ITC));

(**************************************************************************************************************
 	Formatting data
***************************************************************************************************************)

// Fill position
ECR.Position	:= 	F_StuffString(
						InputString 	:= ECR_ITC.Position, 
						StringLength	:= SIS_6_0.POSITION_STRINGLENGTH, 
						StuffCharacter 	:= '0',
						LeftAligned		:= FALSE);

// Fill code
ECR.Code	:= F_StuffString(
					InputString 	:= INT_TO_STRING(ECR_ITC.Code), 
					StringLength	:= SIS_6_0.CONTROLCODE_STRINGLENGTH, 
					StuffCharacter 	:= '0',
					LeftAligned		:= FALSE);

// Fill variable
ECR.Variable 	:= F_StuffString(
					InputString 	:= DINT_TO_STRING(ECR_ITC.Variable), 
					StringLength	:= SIS_6_0.CONTROLVARIABLE_STRINGLENGTH, 
					StuffCharacter 	:= '0',
					LeftAligned		:= FALSE);

// Fill errorcode
ECR.ReturnCode 	:= F_StuffString(
					InputString 	:= INT_TO_STRING(ECR_ITC.ReturnCode), 
					StringLength	:= SIS_6_0.ERRORCODE_STRINGLENGTH, 
					StuffCharacter 	:= '0',
					LeftAligned		:= FALSE);


(**************************************************************************************************************
 	Build string and add to Base Driver
***************************************************************************************************************)
MEMSET(destAddr := ADR(SendTelegram), 0, SIZEOF(SendTelegram));
WritePointer := 0;

F_AssembleByteStream(
	pSrc:= ADR('ECR'), 
	SrcLen:= 3, 
	pDest:= ADR(SendTelegram), 
	DestLen:= SIZEOF(SendTelegram), 
	WritePointer:= WritePointer);

F_AssembleByteStream(
	pSrc:= ADR(ECR.Position), 
	SrcLen:= INT_TO_UDINT(LEN(ECR.Position)), 
	pDest:= ADR(SendTelegram), 
	DestLen:= SIZEOF(SendTelegram), 
	WritePointer:= WritePointer);

F_AssembleByteStream(
	pSrc:= ADR(ECR.Code), 
	SrcLen:= INT_TO_UDINT(LEN(ECR.Code)), 
	pDest:= ADR(SendTelegram), 
	DestLen:= SIZEOF(SendTelegram), 
	WritePointer:= WritePointer);
	
F_AssembleByteStream(
	pSrc:= ADR(ECR.Variable), 
	SrcLen:= INT_TO_UDINT(LEN(ECR.Variable)), 
	pDest:= ADR(SendTelegram), 
	DestLen:= SIZEOF(SendTelegram), 
	WritePointer:= WritePointer);
	
F_AssembleByteStream(
	pSrc:= ADR(ECR.ReturnCode), 
	SrcLen:= INT_TO_UDINT(LEN(ECR.ReturnCode)), 
	pDest:= ADR(SendTelegram), 
	DestLen:= SIZEOF(SendTelegram), 
	WritePointer:= WritePointer);

// Add to buffer of Base Driver
M_ProcessECR := fbBaseDriver.M_SendAppData(
					mpSendData := ADR(SendTelegram),
					mSendDataLen := WritePointer);
					
// Forward to mirror channel
M_MirrorData(Data := ADR(SendTelegram), DataLen := WritePointer);
END_METHOD

METHOD PROTECTED M_ProcessERR : BOOL
(**************************************************************************************
 * 	Application		:	BoxControl Framework
 *	Revision		:	$Revision: 404529 $
 *	Revision date	:	$Date: 2018-04-23 08:21:38 +0200 (Mo., 23 Apr 2018) $
 *	Last changed by	:	$Author: b7bolm $
 *	URL				:	$URL: http://almscdc.swisslog.com/repo/SWPD/Development/BoxControlFramework/20_Release/trunk/01_Software/BCF/BCF/JumpStart/20_Product/10_App/11_Com/10_Lib/10_Conv/12_MFCS/11_SIS/FB_SIS_MsgManager_6_0.TcPOU $
 *
 *	Purpose			:	Send ERR
 *
 * ------------------------------------------------------------------------------------
 *	Copyright Swisslog [IP AG], Switzerland. All rights reserved.
 * 
 * ------------------------------------------------------------------------------------
 *	
 * 	Revision History: 
 *
 * 	VERSION			DATE			INITIALS			DESCRIPTION
 *	0.1				01.01.2001		swl					Example
 *
 **************************************************************************************)
VAR_INPUT
 	meChannelSrc		: E_MFCS_Channel; // Source communicaton channel
	mpERR				: POINTER TO ST_ITC_ERR; // Pointer to ATR
END_VAR
(**************************************************************************************************************
 	Check if a telegram needs to be send
***************************************************************************************************************)
// If settings allow sending a ERR 	
IF  Settings.Telegrams.SendERR THEN
	// If the source of the request is this channel or is undefined
	IF meChannelSrc = Settings.MFCS_Channel OR
		meChannelSrc = E_MFCS_Channel.BEGIN_CHANNEL THEN
		;//Proceed
	ELSE // Source is a different MFCS Connection
		// Dont send a telegram		
		RETURN;
	END_IF	
ELSE
	// Dont send a telegram		
	RETURN;
END_IF

(**************************************************************************************************************
 	ITC - Map generic data to type
***************************************************************************************************************)
MEMCPY(destAddr := ADR(ERR_ITC), srcAddr := mpERR, n := SIZEOF(ERR_ITC));

(**************************************************************************************************************
 	Formatting data
***************************************************************************************************************)
// Fill position
ERR.Position	:= 	F_StuffString(
						InputString 	:= ERR_ITC.Position, 
						StringLength	:= SIS_6_0.POSITION_STRINGLENGTH, 
						StuffCharacter 	:= '0',
						LeftAligned		:= FALSE);

// Fill position
ERR.Code	:= 	F_StuffString(
						InputString 	:= INT_TO_STRING(ERR_ITC.Code), 
						StringLength	:= SIS_6_0.ERR_CODE_STRINGLENGTH, 
						StuffCharacter 	:= '0',
						LeftAligned		:= FALSE);
						
// Get Error Code 
ERR.ReturnCode := F_StuffString(
					InputString 	:= INT_TO_STRING(ERR_ITC.ReturnCode), 
					StringLength	:= SIS_6_0.ERRORCODE_STRINGLENGTH, 
					StuffCharacter 	:= '0',
					LeftAligned		:= FALSE);;
					
(**************************************************************************************************************
 	Build string and add to Base Driver
***************************************************************************************************************)
MEMSET(destAddr := ADR(SendTelegram), 0, SIZEOF(SendTelegram));
WritePointer := 0;

F_AssembleByteStream(
	pSrc:= ADR('ERR'), 
	SrcLen:= 3, 
	pDest:= ADR(SendTelegram), 
	DestLen:= SIZEOF(SendTelegram), 
	WritePointer:= WritePointer);

F_AssembleByteStream(
	pSrc:= ADR(ERR.Position), 
	SrcLen:= INT_TO_UDINT(LEN(ERR.Position)), 
	pDest:= ADR(SendTelegram), 
	DestLen:= SIZEOF(SendTelegram), 
	WritePointer:= WritePointer);

F_AssembleByteStream(
	pSrc:= ADR(ERR.Code), 
	SrcLen:= INT_TO_UDINT(LEN(ERR.Code)), 
	pDest:= ADR(SendTelegram), 
	DestLen:= SIZEOF(SendTelegram), 
	WritePointer:= WritePointer);
	
F_AssembleByteStream(
	pSrc:= ADR(ERR.ReturnCode), 
	SrcLen:= INT_TO_UDINT(LEN(ERR.ReturnCode)), 
	pDest:= ADR(SendTelegram), 
	DestLen:= SIZEOF(SendTelegram), 
	WritePointer:= WritePointer);
	
// Add to buffer of Base Driver
M_ProcessERR := fbBaseDriver.M_SendAppData(
					mpSendData := ADR(SendTelegram),
					mSendDataLen := WritePointer);
					
// Forward to mirror channel
M_MirrorData(Data := ADR(SendTelegram), DataLen := WritePointer);
END_METHOD

METHOD PROTECTED M_ProcessESR : BOOL
(**************************************************************************************
 * 	Application		:	BoxControl Framework
 *	Revision		:	$Revision: 404529 $
 *	Revision date	:	$Date: 2018-04-23 08:21:38 +0200 (Mo., 23 Apr 2018) $
 *	Last changed by	:	$Author: b7bolm $
 *	URL				:	$URL: http://almscdc.swisslog.com/repo/SWPD/Development/BoxControlFramework/20_Release/trunk/01_Software/BCF/BCF/JumpStart/20_Product/10_App/11_Com/10_Lib/10_Conv/12_MFCS/11_SIS/FB_SIS_MsgManager_6_0.TcPOU $
 *
 *	Purpose			:	Send ESR
 *
 * ------------------------------------------------------------------------------------
 *	Copyright Swisslog [IP AG], Switzerland. All rights reserved.
 * 
 * ------------------------------------------------------------------------------------
 *	
 * 	Revision History: 
 *
 * 	VERSION			DATE			INITIALS			DESCRIPTION
 *	0.1				01.01.2001		swl					Example
 *
 **************************************************************************************)
VAR_INPUT
 	meChannelSrc		: E_MFCS_Channel; // Source communicaton channel
	mpESR				: POINTER TO ST_ITC_ESR; // Pointer to ESR
END_VAR
(**************************************************************************************************************
 	Check if a telegram needs to be send
***************************************************************************************************************)
// If settings allow sending a ESR 	
IF  Settings.Telegrams.SendESR THEN
	// If the source of the request is this channel or is undefined
	IF meChannelSrc = Settings.MFCS_Channel OR
		meChannelSrc = E_MFCS_Channel.BEGIN_CHANNEL THEN
		;//Proceed
	ELSE // Source is a different MFCS Connection
		// Dont send a telegram		
		RETURN;
	END_IF	
ELSE
	// Dont send a telegram		
	RETURN;
END_IF

(**************************************************************************************************************
 	ITC - Map generic data to type
***************************************************************************************************************)
MEMCPY(destAddr := ADR(ESR_ITC), srcAddr := mpESR, n := SIZEOF(ESR_ITC));

(**************************************************************************************************************
 	Formatting data
***************************************************************************************************************)
// Build position
ESR.Position := F_StuffString(
					InputString 	:= ESR_ITC.Position, 
					StringLength	:= SIS_6_0.POSITION_STRINGLENGTH, 
					StuffCharacter 	:= '0',
					LeftAligned		:= FALSE);
// Build state
ESR.State := INT_TO_STRING(ESR_ITC.State);

// Build enabled
ESR.Enabled	:= INT_TO_STRING(BOOL_TO_INT(ESR_ITC.Enabled));

// Build error state	
ESR.ErrorState := INT_TO_STRING(ESR_ITC.ErrorState);					

// Build error code
ESR.ErrorCode := F_StuffString(
					InputString 	:= INT_TO_STRING(ESR_ITC.ErrorCode), 
					StringLength	:= SIS_6_0.ERRORCODE_STRINGLENGTH, 
					StuffCharacter 	:= '0',
					LeftAligned		:= FALSE);
					
// Build error type
ESR.ErrorType := INT_TO_STRING(ESR_ITC.ErrorType);

// Build information
ESR.ErrorInformation := F_StuffString(
							InputString 	:= ESR_ITC.ErrorInformation, 
							StringLength	:= SIS_6_0.ERRORINFORMATION_STRINGLENGTH, 
							StuffCharacter 	:= ' ',
							LeftAligned		:= TRUE);
// Build variable
ESR.Variable  := F_StuffString(
					InputString 	:= DINT_TO_STRING(ESR_ITC.Variable), 
					StringLength	:= SIS_6_0.CONTROLVARIABLE_STRINGLENGTH, 
					StuffCharacter 	:= '0',
					LeftAligned		:= FALSE);

// Get Error Code 
ESR.ReturnCode := F_StuffString(
					InputString 	:= INT_TO_STRING(ESR_ITC.ReturnCode), 
					StringLength	:= SIS_6_0.ERRORCODE_STRINGLENGTH, 
					StuffCharacter 	:= '0',
					LeftAligned		:= FALSE);

(**************************************************************************************************************
 	Build string and add to Base Driver
***************************************************************************************************************)
MEMSET(destAddr := ADR(SendTelegram), 0, SIZEOF(SendTelegram));
WritePointer := 0;

F_AssembleByteStream(
	pSrc:= ADR('ESR'), 
	SrcLen:= 3, 
	pDest:= ADR(SendTelegram), 
	DestLen:= SIZEOF(SendTelegram), 
	WritePointer:= WritePointer);
	
F_AssembleByteStream(
	pSrc:= ADR(ESR.Position), 
	SrcLen:= INT_TO_UDINT(LEN(ESR.Position)), 
	pDest:= ADR(SendTelegram), 
	DestLen:= SIZEOF(SendTelegram), 
	WritePointer:= WritePointer);
	
F_AssembleByteStream(
	pSrc:= ADR(ESR.State), 
	SrcLen:= INT_TO_UDINT(LEN(ESR.State)), 
	pDest:= ADR(SendTelegram), 
	DestLen:= SIZEOF(SendTelegram), 
	WritePointer:= WritePointer);	
	
F_AssembleByteStream(
	pSrc:= ADR(ESR.Enabled), 
	SrcLen:= INT_TO_UDINT(LEN(ESR.Enabled)), 
	pDest:= ADR(SendTelegram), 
	DestLen:= SIZEOF(SendTelegram), 
	WritePointer:= WritePointer);	


F_AssembleByteStream(
	pSrc:= ADR(ESR.ErrorState), 
	SrcLen:= INT_TO_UDINT(LEN(ESR.ErrorState)), 
	pDest:= ADR(SendTelegram), 
	DestLen:= SIZEOF(SendTelegram), 
	WritePointer:= WritePointer);		

F_AssembleByteStream(
	pSrc:= ADR(ESR.ErrorCode), 
	SrcLen:= INT_TO_UDINT(LEN(ESR.ErrorCode)), 
	pDest:= ADR(SendTelegram), 
	DestLen:= SIZEOF(SendTelegram), 
	WritePointer:= WritePointer);	

F_AssembleByteStream(
	pSrc:= ADR(ESR.ErrorType), 
	SrcLen:= INT_TO_UDINT(LEN(ESR.ErrorType)), 
	pDest:= ADR(SendTelegram), 
	DestLen:= SIZEOF(SendTelegram), 
	WritePointer:= WritePointer);		
	
F_AssembleByteStream(
	pSrc:= ADR(ESR.ErrorInformation), 
	SrcLen:= INT_TO_UDINT(LEN(ESR.ErrorInformation)), 
	pDest:= ADR(SendTelegram), 
	DestLen:= SIZEOF(SendTelegram), 
	WritePointer:= WritePointer);	
	
F_AssembleByteStream(
	pSrc:= ADR(ESR.Variable), 
	SrcLen:= INT_TO_UDINT(LEN(ESR.Variable)), 
	pDest:= ADR(SendTelegram), 
	DestLen:= SIZEOF(SendTelegram), 
	WritePointer:= WritePointer);	

F_AssembleByteStream(
	pSrc:= ADR(ESR.ReturnCode), 
	SrcLen:= INT_TO_UDINT(LEN(ESR.ReturnCode)), 
	pDest:= ADR(SendTelegram), 
	DestLen:= SIZEOF(SendTelegram), 
	WritePointer:= WritePointer);		

// Add to buffer of Base Driver
M_ProcessESR := fbBaseDriver.M_SendAppData(
					mpSendData := ADR(SendTelegram),
					mSendDataLen := WritePointer);

// Forward to mirror channel
M_MirrorData(Data := ADR(SendTelegram), DataLen := WritePointer);
END_METHOD

